(* Logix 5000 project; controller WWTP_SEC_CLX vendor 1 type 14 code 54 rev 17.2; software revision 17.00; part 8 of 13 *)
(* tags used below, declared in another part *)
   Wrk_FirstColdStartT : TIMER;   // Time since first cold start
   Wrk_FirstFailColdT : TIMER;   // Time for cold motor to wait after 1st start failure before ready
   Wrk_SubsFailColdT : TIMER;   // Time for cold motor to wait after 2nd and subs. failures before ready
   Wrk_FirstFailHotT : TIMER;   // Time for hot motor to wait after 1st start failure before ready
   Wrk_SubsFailHotT : TIMER;   // Time for hot motor to wait after 2nd and subs. failures before ready
   Wrk_HotRestartOKT : TIMER;   // Time for hot motor to run so it can restart immediately when stopped
   Wrk_RestartHotT : TIMER;   // Time for hot motor to wait after stop after running less than Hot Restart OK time
   Wrk_HotToColdT : TIMER;   // Time for a stopped hot motor to become cold
   Wrk_State : DINT;   // Instruction State (see state diagram in design docs)
   Wrk_SecondColdStartT : TIMER;   // Time since second cold start
(* P_ResInh, continued *)

ROUTINE Prescan   (* ladder *)
// Clear timers and set to known state
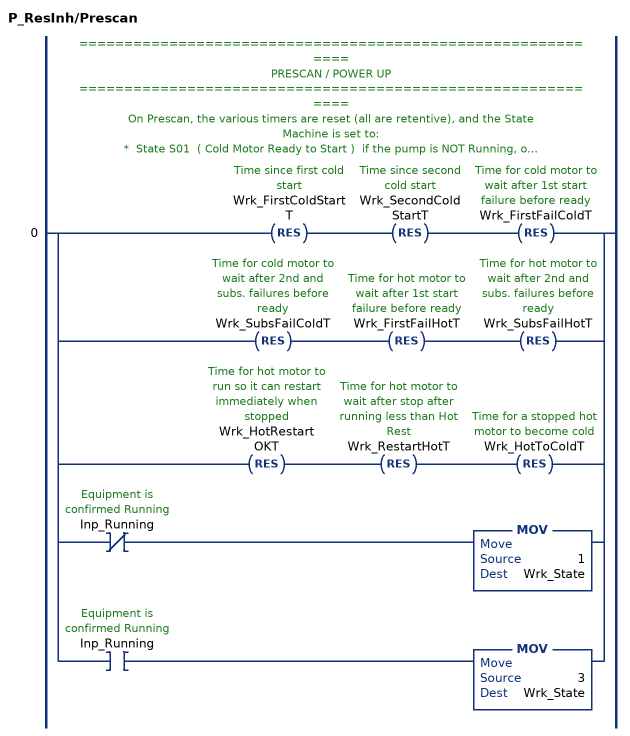
   // ============================================================
   // PRESCAN / POWER UP
   // ============================================================
   // On Prescan, the various timers are reset (all are retentive), and the State
   // Machine is set to:
   // *  State S01  ( Cold Motor Ready to Start )  if the pump is NOT Running, or
   // *  State S03  ( Cold Motor Running )  if the pump is Running.
   0: [RES(Wrk_FirstColdStartT) RES(Wrk_SecondColdStartT) RES(Wrk_FirstFailColdT) ,RES(Wrk_SubsFailColdT) RES(Wrk_FirstFailHotT) RES(Wrk_SubsFailHotT) ,RES(Wrk_HotRestartOKT) RES(Wrk_RestartHotT) RES(Wrk_HotToColdT) ,XIO(Inp_Running) MOV(1,Wrk_State) ,XIC(Inp_Running) MOV(3,Wrk_State) ];
END_ROUTINE
END_ADD_ON_INSTRUCTION

ADD_ON_INSTRUCTION P_RunTime   (* revision 0.7, ExecutePrescan, ExecuteEnableInFalse *)
// Run Time and Starts
// Revision note:
// Aligned name, description and local STRING values, sizes, across instructions.
// Help:
// This Instruction monitors the "Running" and "Starting" Status of a motor or other device and  provides:
// *  Total accumulated run time, in 1/10 hour increments (hour meter)
// *  Total number of starts or start attemptes (count)
// *  Maximum continuous run time for any start (hours)
// *  Program and Maintenance Commands to allow clearing of the totals/maximum
VAR_INPUT
   Inp_Starting : BOOL; {visible}   // 1=Motor is Starting (from motor instruction)
   Inp_Running : BOOL := 1; {visible}   // 1=Motor is Running (from motor instruction)
   Cfg_PCmdClear : BOOL := 1;   // 1=Clear Program Commands on receipt 0=Leave Set
   PCmd_ClearStarts : BOOL;   // Program Command to Clear Count of Starts (attempts)
   PCmd_ClearMaxHrs : BOOL;   // Program Command to Clear Maximum (continuous) Run Time for any start
   PCmd_ClearTotHrs : BOOL;   // Program Command to Clear Total Running Time
   MCmd_ClearStarts : BOOL;   // Maintenance Command to Clear Count of Starts (attempts)
   MCmd_ClearMaxHrs : BOOL;   // Maintenance Command to Clear Maximum (continuous) Run Time for any start
   MCmd_ClearTotHrs : BOOL;   // Maintenance Command to Clear Total Running Time
END_VAR
VAR_OUTPUT
   Val_Starts : DINT; {visible}   // Total number of motor starts or attempts
   Val_CurRunHrs : REAL; {visible}   // Current running time this start (hours)
   Val_MaxRunHrs : REAL; {visible}   // Maximum continuous running time for a given start (hours)
   Val_TotRunHrs : REAL; {visible}   // Total accumulated running time (hours)
END_VAR
VAR
   Wrk_CurHours : DINT;   // Whole hours of current run time
   Wrk_CurRunT : TIMER := (PRE := 2147483647);   // Timer for timing current run time
   Wrk_TotTenths : DINT;   // Tenths of hours of total run time
   Wrk_Starts : COUNTER := (PRE := 2147483647);   // Counter for counting motor starts
   Wrk_TotRunT : TIMER := (PRE := 2147483647);   // Retentive timer for timing 0.1 hour total run time
   Wrk_MaxHours : REAL;   // Internal Maximum Run Hours
END_VAR

ROUTINE EnableInFalse   (* ladder *)
// False Rung or Enable In False: as if motor is Stopped
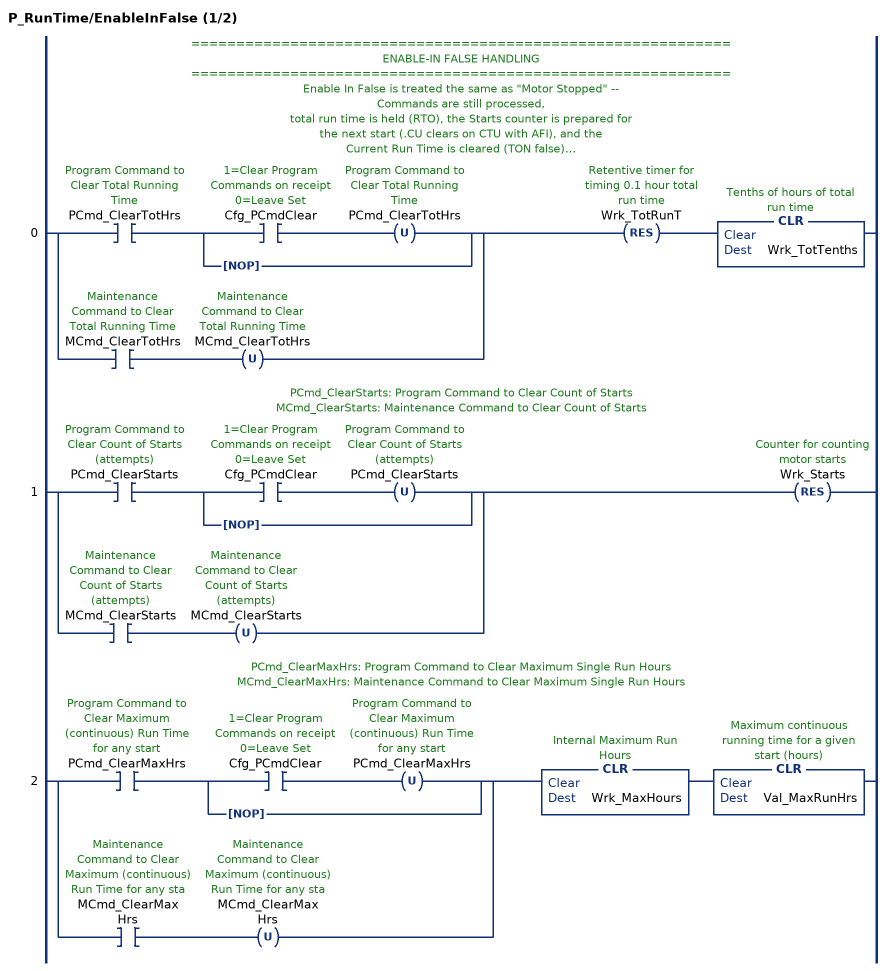
   // ============================================================
   // ENABLE-IN FALSE HANDLING
   // ============================================================
   // Enable In False is treated the same as "Motor Stopped" --
   // Commands are still processed,
   // total run time is held (RTO), the Starts counter is prepared for
   // the next start (.CU clears on CTU with AFI), and the
   // Current Run Time is cleared (TON false).
   // ============================================================
   // COMMAND PROCESSING
   // ============================================================
   // These rungs handle received Commands.  This object has no Modes and
   // Commands are accepted regardless of Mode.  Commands should be
   // restricted to authorized personnel (typically at a maintenance level).
   // PCmd_ClearTotHrs: Program Command to Clear Total Runtime Hours
   // MCmd_ClearTotHrs: Maintenance Command to Clear Total Runtime Hours
   0: [XIC(PCmd_ClearTotHrs) [XIC(Cfg_PCmdClear) OTU(PCmd_ClearTotHrs) ,NOP() ] ,XIC(MCmd_ClearTotHrs) OTU(MCmd_ClearTotHrs) ]RES(Wrk_TotRunT)CLR(Wrk_TotTenths);
   // PCmd_ClearStarts: Program Command to Clear Count of Starts
   // MCmd_ClearStarts: Maintenance Command to Clear Count of Starts
   1: [XIC(PCmd_ClearStarts) [XIC(Cfg_PCmdClear) OTU(PCmd_ClearStarts) ,NOP() ] ,XIC(MCmd_ClearStarts) OTU(MCmd_ClearStarts) ]RES(Wrk_Starts);
   // PCmd_ClearMaxHrs: Program Command to Clear Maximum Single Run Hours
   // MCmd_ClearMaxHrs: Maintenance Command to Clear Maximum Single Run Hours
   2: [XIC(PCmd_ClearMaxHrs) [XIC(Cfg_PCmdClear) OTU(PCmd_ClearMaxHrs) ,NOP() ] ,XIC(MCmd_ClearMaxHrs) OTU(MCmd_ClearMaxHrs) ]CLR(Wrk_MaxHours)CLR(Val_MaxRunHrs);
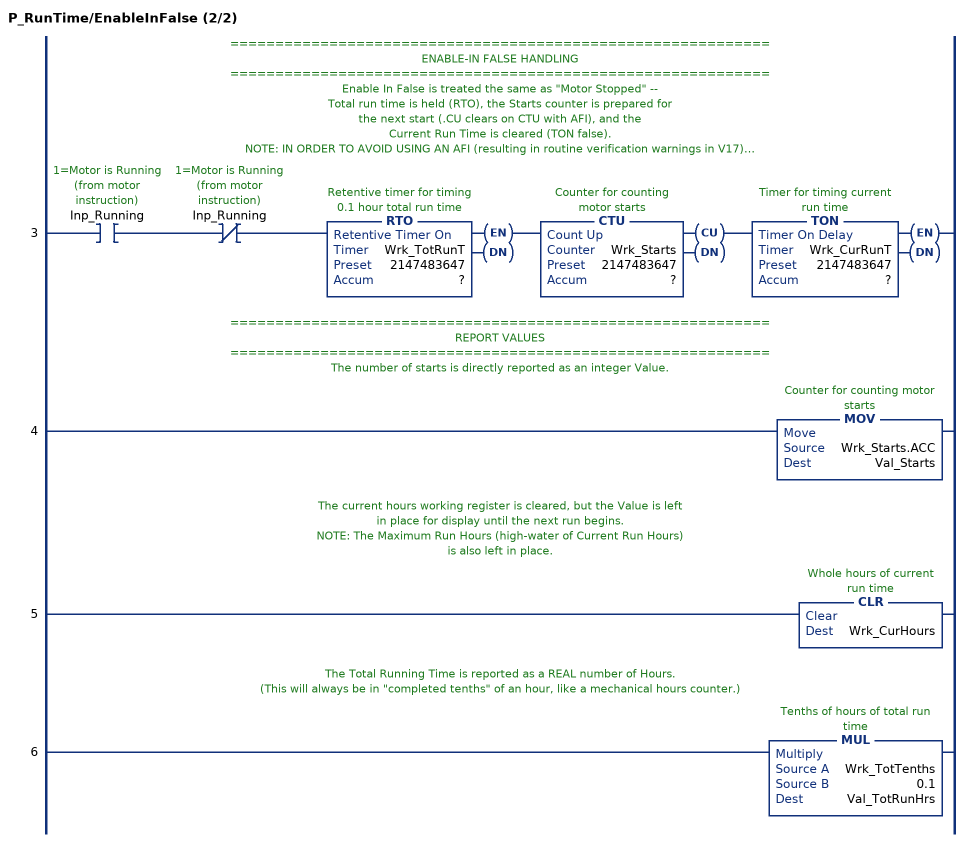
   // ============================================================
   // ENABLE-IN FALSE HANDLING
   // ============================================================
   // Enable In False is treated the same as "Motor Stopped" --
   // Total run time is held (RTO), the Starts counter is prepared for
   // the next start (.CU clears on CTU with AFI), and the
   // Current Run Time is cleared (TON false).
   // NOTE: IN ORDER TO AVOID USING AN AFI (resulting in routine verification warnings in V17),
   // THIS RUNG USES AN XIC AND XIO OF THE SAME BIT TO ENSURE THE
   // TIMERS AND COUNTER ARE SCANNED FALSE.
   // THIS IS NOT DEAD CODE.  IT IS INTENTIONALLY CODED THIS WAY FOR PROPER OPERATION.
   3: XIC(Inp_Running)XIO(Inp_Running)RTO(Wrk_TotRunT,?,?)CTU(Wrk_Starts,?,?)TON(Wrk_CurRunT,?,?);
   // ============================================================
   // REPORT VALUES
   // ============================================================
   // The number of starts is directly reported as an integer Value.
   4: MOV(Wrk_Starts.ACC,Val_Starts);
   // The current hours working register is cleared, but the Value is left
   // in place for display until the next run begins.
   // NOTE: The Maximum Run Hours (high-water of Current Run Hours)
   // is also left in place.
   5: CLR(Wrk_CurHours);
   // The Total Running Time is reported as a REAL number of Hours.
   // (This will always be in "completed tenths" of an hour, like a mechanical hours counter.)
   6: MUL(Wrk_TotTenths,0.1,Val_TotRunHrs);
END_ROUTINE

ROUTINE Logic   (* ladder *)
// Accumulate Run Time (if runnings) and Count Starts
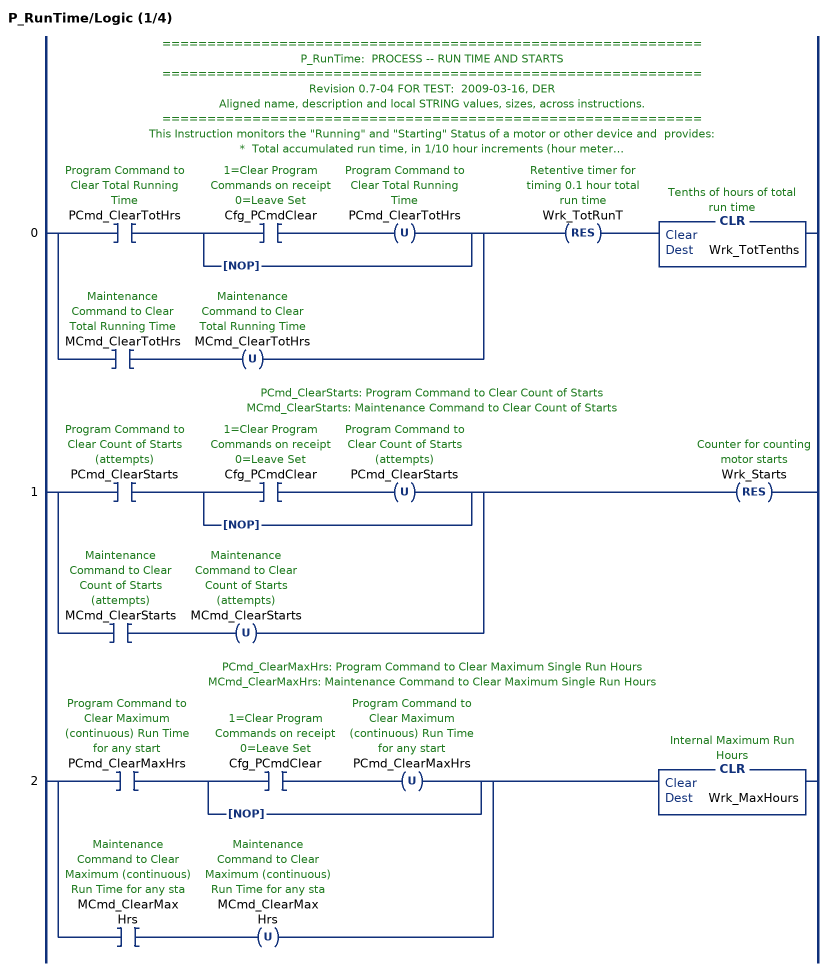
   // ============================================================
   // P_RunTime:  PROCESS -- RUN TIME AND STARTS
   // ============================================================
   // Revision 0.7-04 FOR TEST:  2009-03-16, DER
   // Aligned name, description and local STRING values, sizes, across instructions.
   // ============================================================
   // This Instruction monitors the "Running" and "Starting" Status of a motor or other device and  provides:
   // *  Total accumulated run time, in 1/10 hour increments (hour meter)
   // *  Total number of starts or start attemptes (count)
   // *  Maximum continuous run time for any start (hours)
   // * Commands to allow clearing of the totals/maximum
   // ============================================================
   // COMMAND PROCESSING
   // ============================================================
   // These rungs handle received Commands.  This object has no Modes and
   // Commands are accepted regardless of Mode.  Commands should be
   // restriceted to authorized personnel (typically at a maintenance level).
   // PCmd_ClearTotHrs: Program Command to Clear Total Runtime Hours
   // MCmd_ClearTotHrs: Maintenance Command to Clear Total Runtime Hours
   0: [XIC(PCmd_ClearTotHrs) [XIC(Cfg_PCmdClear) OTU(PCmd_ClearTotHrs) ,NOP() ] ,XIC(MCmd_ClearTotHrs) OTU(MCmd_ClearTotHrs) ]RES(Wrk_TotRunT)CLR(Wrk_TotTenths);
   // PCmd_ClearStarts: Program Command to Clear Count of Starts
   // MCmd_ClearStarts: Maintenance Command to Clear Count of Starts
   1: [XIC(PCmd_ClearStarts) [XIC(Cfg_PCmdClear) OTU(PCmd_ClearStarts) ,NOP() ] ,XIC(MCmd_ClearStarts) OTU(MCmd_ClearStarts) ]RES(Wrk_Starts);
   // PCmd_ClearMaxHrs: Program Command to Clear Maximum Single Run Hours
   // MCmd_ClearMaxHrs: Maintenance Command to Clear Maximum Single Run Hours
   2: [XIC(PCmd_ClearMaxHrs) [XIC(Cfg_PCmdClear) OTU(PCmd_ClearMaxHrs) ,NOP() ] ,XIC(MCmd_ClearMaxHrs) OTU(MCmd_ClearMaxHrs) ]CLR(Wrk_MaxHours);
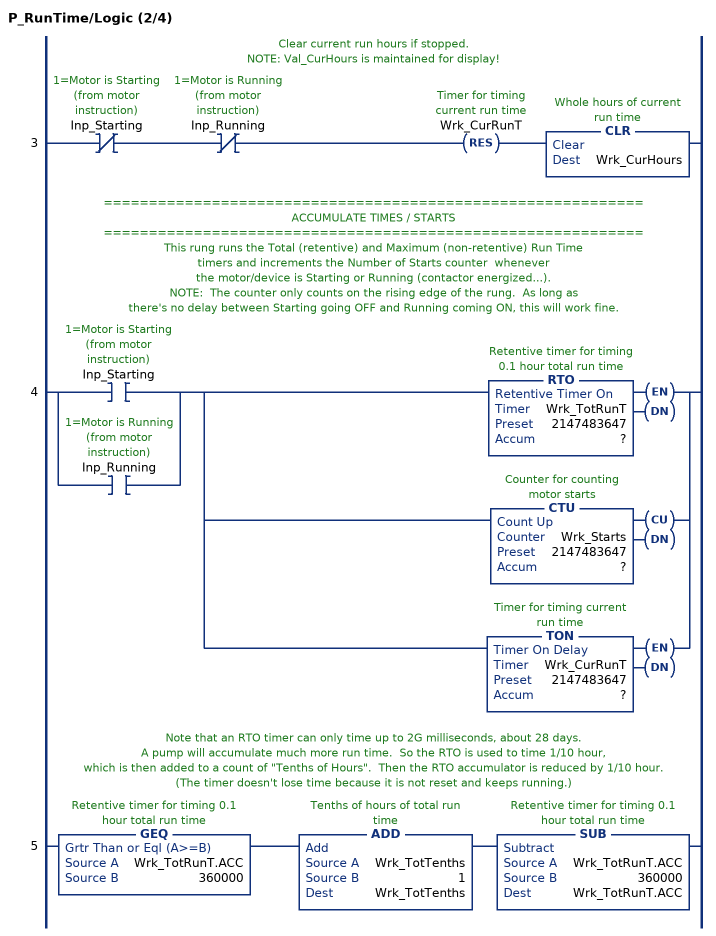
   // Clear current run hours if stopped.
   // NOTE: Val_CurHours is maintained for display!
   3: XIO(Inp_Starting)XIO(Inp_Running)RES(Wrk_CurRunT)CLR(Wrk_CurHours);
   // ============================================================
   // ACCUMULATE TIMES / STARTS
   // ============================================================
   // This rung runs the Total (retentive) and Maximum (non-retentive) Run Time
   // timers and increments the Number of Starts counter  whenever
   //  the motor/device is Starting or Running (contactor energized...).
   // NOTE:  The counter only counts on the rising edge of the rung.  As long as
   // there's no delay between Starting going OFF and Running coming ON, this will work fine.
   4: [XIC(Inp_Starting) ,XIC(Inp_Running) ][RTO(Wrk_TotRunT,?,?) ,CTU(Wrk_Starts,?,?) ,TON(Wrk_CurRunT,?,?) ];
   // Note that an RTO timer can only time up to 2G milliseconds, about 28 days.
   // A pump will accumulate much more run time.  So the RTO is used to time 1/10 hour,
   // which is then added to a count of "Tenths of Hours".  Then the RTO accumulator is reduced by 1/10 hour.
   // (The timer doesn't lose time because it is not reset and keeps running.)
   5: GEQ(Wrk_TotRunT.ACC,360000)ADD(Wrk_TotTenths,1,Wrk_TotTenths)SUB(Wrk_TotRunT.ACC,360000,Wrk_TotRunT.ACC);
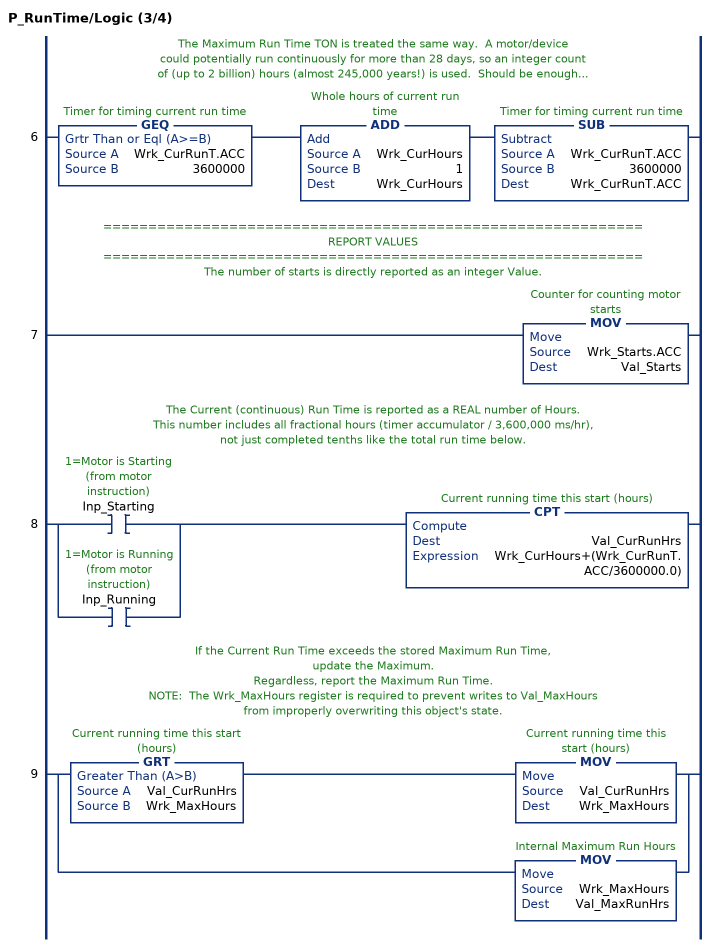
   // The Maximum Run Time TON is treated the same way.  A motor/device
   // could potentially run continuously for more than 28 days, so an integer count
   // of (up to 2 billion) hours (almost 245,000 years!) is used.  Should be enough...
   6: GEQ(Wrk_CurRunT.ACC,3600000)ADD(Wrk_CurHours,1,Wrk_CurHours)SUB(Wrk_CurRunT.ACC,3600000,Wrk_CurRunT.ACC);
   // ============================================================
   // REPORT VALUES
   // ============================================================
   // The number of starts is directly reported as an integer Value.
   7: MOV(Wrk_Starts.ACC,Val_Starts);
   // The Current (continuous) Run Time is reported as a REAL number of Hours.
   // This number includes all fractional hours (timer accumulator / 3,600,000 ms/hr),
   // not just completed tenths like the total run time below.
   8: [XIC(Inp_Starting) ,XIC(Inp_Running) ]CPT(Val_CurRunHrs,Wrk_CurHours+(Wrk_CurRunT.ACC/3600000.0));
   // If the Current Run Time exceeds the stored Maximum Run Time,
   // update the Maximum.
   // Regardless, report the Maximum Run Time.
   // NOTE:  The Wrk_MaxHours register is required to prevent writes to Val_MaxHours
   // from improperly overwriting this object's state.
   9: [GRT(Val_CurRunHrs,Wrk_MaxHours) MOV(Val_CurRunHrs,Wrk_MaxHours) ,MOV(Wrk_MaxHours,Val_MaxRunHrs) ];
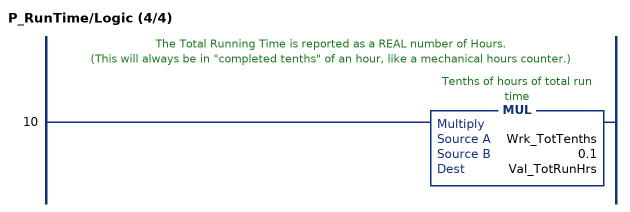
   // The Total Running Time is reported as a REAL number of Hours.
   // (This will always be in "completed tenths" of an hour, like a mechanical hours counter.)
   10: MUL(Wrk_TotTenths,0.1,Val_TotRunHrs);
END_ROUTINE

ROUTINE Prescan   (* ladder *)
// Set Current Run time internally to 0.  Display value is left in place.
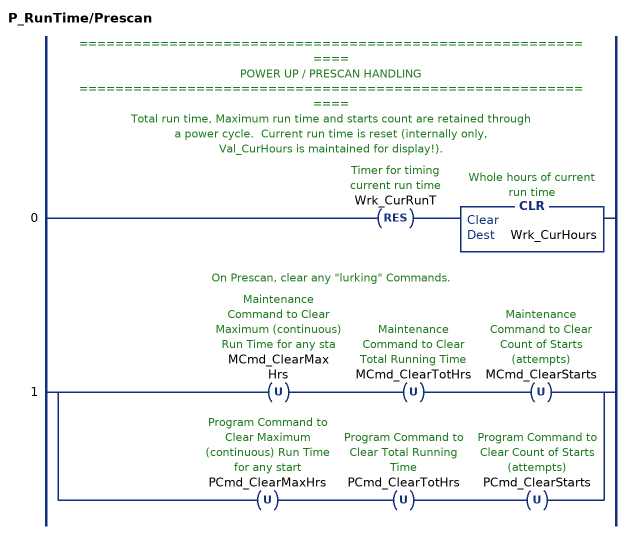
   // ============================================================
   // POWER UP / PRESCAN HANDLING
   // ============================================================
   // Total run time, Maximum run time and starts count are retained through
   // a power cycle.  Current run time is reset (internally only,
   // Val_CurHours is maintained for display!).
   0: RES(Wrk_CurRunT)CLR(Wrk_CurHours);
   // On Prescan, clear any "lurking" Commands.
   1: [OTU(MCmd_ClearMaxHrs) OTU(MCmd_ClearTotHrs) OTU(MCmd_ClearStarts) ,OTU(PCmd_ClearMaxHrs) OTU(PCmd_ClearTotHrs) OTU(PCmd_ClearStarts) ];
END_ROUTINE
END_ADD_ON_INSTRUCTION

ADD_ON_INSTRUCTION P_VSD   (* revision 0.15, ExecutePrescan, ExecuteEnableInFalse *)
// Variable Speed Drive
// Revision note:
// Aligned name, description and local STRING values, sizes, across instructions.
// Help:
// This Instruction controls and monitors a Variable-Speed (AC or DC) Drive
// and provides:
// *  Starting drive, stopping drive, jogging drive, setting speed reference and setting direction
// *  Monitoring of run feedback, display of actual drive status, including accel, decel, direction, speed
// *  Detection of Failure to Start, Failure to Stop, Drive Fault/Not Ready
// *  Monitoring of Permissive conditions to allow starting
// *  Monitoring of Interlock conditions to stop drive or prevent starting
// *  Simulation, providing feedback of a working drive while disabling outputs
// *  Monitoring of I/O communication faults
// *  Alarms for Fail to Start, Fail to Stop, Interlock Trip, Drive Fault/Not Ready, I/O Fault
// *  Operation in Hand, Maintenance, Override, Program and Operator Modes
// *  "Available" status for use by automation logic to know whether drive
//       can be controlled by other objects.
VAR_INPUT
   Inp_SpeedFdbk : INT; {visible}   // Speed Feedbak in Drive Units (typ. 0-32767 = 0 to max freq.)
   Inp_FaultCode : INT;   // Current Drive Fault Code (enumeration)
   Inp_Datalink : INT; {visible}   // Auxiliary Signal (datalink) Input in Drive (raw) Units
   Inp_Ready : BOOL := 1; {visible}   // 1=Drive is ready to run
   Inp_Running : BOOL; {visible}   // 1=Drive is Running (active)
   Inp_CommandDir : BOOL := 1; {visible}   // 1=Drive is commanded Forward, 0=Drive is commanded Reverse
   Inp_ActualDir : BOOL := 1; {visible}   // 1=Drive is running Forward, 0=Drive is running Reverse
   Inp_Accelerating : BOOL; {visible}   // 1=Drive is accelerating
   Inp_Decelerating : BOOL; {visible}   // 1=Drive is decelerating
   Inp_Alarm : BOOL; {visible}   // 1=Drive has an Alarm Condition (see drive display or manual)
   Inp_Faulted : BOOL; {visible}   // 1=Drive has Faulted (see drive display or manual)
   Inp_AtSpeed : BOOL; {visible}   // 1=Drive is at commanded speed
   Inp_FwdPermOK : BOOL := 1; {visible}   // 1=Permissives OK, drive can start Forward
   Inp_FwdNBPermOK : BOOL := 1; {visible}   // 1=Non-Bypassable Permissives OK, drive can start Forward
   Inp_RevPermOK : BOOL := 1; {visible}   // 1=Permissives OK, drive can start Reverse
   Inp_RevNBPermOK : BOOL := 1; {visible}   // 1=Non-Bypassable Permissives OK, motor can start Reverse
   Inp_IntlkOK : BOOL := 1; {visible}   // 1=Interlocks OK, drive can start/run
   Inp_NBIntlkOK : BOOL := 1; {visible}   // 1=Non-Bypassable Interlocks OK, drive can start/run
   Inp_IOFault : BOOL;   // Input Communication Status 0=OK, 1=fail
   Inp_Sim : BOOL;   // 1=Simulate working drive; 0=Start/Stop/ Monitor actual drive
   Inp_Hand : BOOL; {visible}   // 1=Select Hand (hardwired) Control Strategy
   Inp_Ovrd : BOOL; {visible}   // 1=Select Override control strategy
   Inp_OvrdState : BOOL; {visible}   // 1=Override to RUN, 0=Override to STOP
   Inp_OvrdSpeed : REAL; {visible}   // Speed at which to run drive in Override if Overriding to RUN
   Inp_Reset : BOOL; {visible}   // 1=Reset drive fault conditions and latched Alarms
   Cfg_HasReverse : BOOL;   // 1=Drive can be run reverse, 0=Forward only
   Cfg_HasJog : BOOL;   // 1=Drive Jog Command enabled/visible, 0=Drive Jog Command not allowed
   Cfg_HasRunFdbk : BOOL := 1;   // 1=Drive provides speed feedback and run signal
   Cfg_UseRunFdbk : BOOL := 1;   // 1=Drive run feedback should be used for failure checking
   Cfg_HasInpDatalink : BOOL;   // 1=A signal is connected to Inp_Datalink1
   Cfg_HasOutDatalink : BOOL;   // 1=A signal is connected to Out_Datalink1
   Cfg_HasFwdPermObj : BOOL;   // 1=Tells HMI a P_Perm is connected to Inp_FwdPerm
   Cfg_HasRevPermObj : BOOL;   // 1=Tells HMI a P_Perm is connected to Inp_RevPerm
   Cfg_HasIntlkObj : BOOL;   // 1=Tells HMI a P_Intlk is connected to Inp_Intlk
   Cfg_HasResInhObj : BOOL;   // 1=Tells HMI a P_ResInh Restart Inhibit is connected
   Cfg_HasRunTimeObj : BOOL;   // 1=Tells HMI a P_RunTime is connected
   Cfg_SetTrack : BOOL := 1;   // 1=PSets track OSets in Oper, OSets track PSets in Prog, 0=no tracking
   Cfg_SetTrackOvrdHand : BOOL;   // 1=Prog/Oper Settings track Override/Hand speed reference
   Cfg_PCmdClear : BOOL := 1;   // 1=Clear Program Commands on receipt 0=Leave Set
   Cfg_OvrdPermIntlk : BOOL;   // 1=Override ignores Bypassable Perm/ Intlk; 0=always use Perm/Intlk
   Cfg_HasFailToStartAlm : BOOL;   // 1=Fail to Start Alarm exists and will be checked
   Cfg_HasFailToStopAlm : BOOL;   // 1=Fail to Stop Alarm exists and will be checked
   Cfg_HasIntlkTripAlm : BOOL;   // 1=Interlock Trip Alarm exists and will be checked
   Cfg_HasDriveFaultAlm : BOOL;   // 1=Drive Fault alarm exists and will be checked
   Cfg_HasIOFaultAlm : BOOL;   // 1=I/O Fault Alarm exists and will be checked
   Cfg_FailToStartResetReqd : BOOL;   // 1=Reset requied to clear Fail to Start Alarm
   Cfg_FailToStopResetReqd : BOOL;   // 1=Reset required to clear Fail to Stop Alarm
   Cfg_IntlkTripResetReqd : BOOL;   // 1=Reset required to clear Interlock Trip Alarm
   Cfg_DriveFaultResetReqd : BOOL := 1;   // 1=Reset required to clear Drive Fault Alarm
   Cfg_IOFaultResetReqd : BOOL;   // 1=Reset required to clear I/O Fault Alarm
   Cfg_FailToStartAckReqd : BOOL := 1;   // 1=Acknowledge required for Fail to Start Alarm
   Cfg_FailToStopAckReqd : BOOL := 1;   // 1=Acknowledge required for Fail to Stop Alarm
   Cfg_IntlkTripAckReqd : BOOL := 1;   // 1=Acknowledge required for Interlock Trip Alarm
   Cfg_DriveFaultAckReqd : BOOL;   // 1=Acknowledge required for Drive Fault Alarm
   Cfg_IOFaultAckReqd : BOOL := 1;   // 1=Acknowledge required for I/O Fault Alarm
   Cfg_FailToStartSeverity : SINT := 4;   // Fail To Start Alarm Severity 1=info 2=warn 3=excep 4=fault
   Cfg_FailToStopSeverity : SINT := 4;   // Fail To Stop Alarm Severity 1=info 2=warn 3=excep 4=fault
   Cfg_IntlkTripSeverity : SINT := 2;   // Interlock Trip Alarm Severity 1=info 2=warn 3=excep 4=fault
   Cfg_DriveFaultSeverity : SINT := 4;   // Drive Fault Alarm Severity 1=info, 2=warn, 3=excep, 4=fault
   Cfg_IOFaultSeverity : SINT := 4;   // I/O Fault Alarm Severity 1=info 2=warn 3=excep 4=fault
   Cfg_MinSpdRef : REAL;   // Minimum Speed Reference in EU (for limiting)
   Cfg_MaxSpdRef : REAL := 60.0;   // Maximum Speed Reference in EU (for limiting)
   Cfg_SpeedRefRawMin : INT;   // Speed Reference Minimum in Drive (raw) Units (for scaling)
   Cfg_SpeedRefRawMax : INT := 32767;   // Speed Reference Maximum in Drive (raw) Units (for scaling)
   Cfg_SpeedRefEUMin : REAL;   // Speed Reference Minimum in Engineering Units (for scaling)
   Cfg_SpeedRefEUMax : REAL := 130.0;   // Speed Reference Maximum in Engineering Units (for scaling)
   Cfg_SpeedFdbkRawMin : INT;   // Speed Feedback Minimum in Drive (raw) Units (for scaling)
   Cfg_SpeedFdbkRawMax : INT := 32767;   // Speed Feedback Maximum in Drive (raw) Units (for scaling)
   Cfg_SpeedFdbkEUMin : REAL;   // Speed Feedback Minimum in Engineering Units (for scaling)
   Cfg_SpeedFdbkEUMax : REAL := 130.0;   // Speed Feedback Maximum in Engineering Units (for scaling)
   Cfg_InpDatalinkRawMin : INT;   // Input Datalink Minimum in Drive (raw) Units (for scaling)
   Cfg_InpDatalinkRawMax : INT := 4095;   // Input Datalink Maximum in Drive (raw) Units (for scaling)
   Cfg_InpDatalinkEUMin : REAL;   // Input Datalink Minimum in Engineering Units (for scaling)
   Cfg_InpDatalinkEUMax : REAL := 409.5;   // Input Datalink Maximum in Engineering Units (for scaling)
   Cfg_OutDatalinkMin : REAL;   // Minimum Output Datalink in EU (for limiting)
   Cfg_OutDatalinkMax : REAL := 100.0;   // Maximum Output Datalink in EU (for limiting)
   Cfg_OutDatalinkRawMin : INT;   // Output Datalink Minimum in Drive (raw) Units (for scaling)
   Cfg_OutDatalinkRawMax : INT := 4095;   // Output Datalink Maximum in Drive (raw) Units (for scaling)
   Cfg_OutDatalinkEUMin : REAL;   // Output Datalink Minimum in Engineering Units (for scaling)
   Cfg_OutDatalinkEUMax : REAL := 409.5;   // Output Datalink Maximum in Engineering Units (for scaling)
   Cfg_SimRampT : DINT := 10;   // Time to ramp speed fdbk when in Simulation (sec)
   Cfg_FailToStartT : DINT := 15;   // Time after Start to get Run Feedback before Fault (sec)
   Cfg_FailToStopT : DINT := 15;   // Time after Stop to drop Run Feedback before Fault (sec)
   Cfg_ResetPulseT : DINT := 2;   // Time to pulse Out_Reset to clear drive fault
   PSet_SpeedRef : REAL;   // Program Setting of Speed Reference (EU)
   PSet_OutDatalink : REAL;   // Program Setting of Output Datalink (EU)
   PSet_Owner : DINT;   // Program Owner Request ID (non-zero) or Release (zero)
   OSet_SpeedRef : REAL;   // Operator Setting of Speed Reference (EU)
   OSet_OutDatalink : REAL;   // Operator Setting of Output Datalink (EU)
   PCmd_Start : BOOL;   // Program Command to Start Drive
   PCmd_Stop : BOOL;   // Program Command to Stop Drive
   PCmd_Fwd : BOOL;   // Program Command to set direction to Fowrard
   PCmd_Rev : BOOL;   // Program Command to set direction to Reverse
   PCmd_Acq : BOOL;   // Program Command to Acquire ownership (Oper/OOS to Prog)
   PCmd_Rel : BOOL;   // Program Command to Release ownership (Prog to OOS)
   PCmd_Lock : BOOL;   // Program Command to Lock Mode in Prog
   PCmd_Unlock : BOOL;   // Program Command to Unlock Mode
   PCmd_Reset : BOOL;   // Program Command to Reset drive fault and all Alarms requiring Reset
   PCmd_FailToStartAck : BOOL;   // Program Command to Acknowledge Fail to Start Alarm
   PCmd_FailToStartInhibit : BOOL;   // Program Command to Inhibit Fail to Start Alarm
   PCmd_FailToStartUninhibit : BOOL;   // Program Command to Uninhibit Fail to Start Alarm
   PCmd_FailToStopAck : BOOL;   // Program Command to Acknowledge Fail to Stop Alarm
   PCmd_FailToStopInhibit : BOOL;   // Program Command to Inhibit Fail to Stop Alarm
   PCmd_FailToStopUninhibit : BOOL;   // Program Command to Uninhibit Fail to Stop Alarm
   PCmd_IntlkTripAck : BOOL;   // Program Command to Acknowledge Interlock Trip Alarm
   PCmd_IntlkTripInhibit : BOOL;   // Program Command to Inhibit Interlock Trip Alarm
   PCmd_IntlkTripUninhibit : BOOL;   // Program Command to Uninhibit Interlock Trip Alarm
   PCmd_DriveFaultAck : BOOL;   // Program Command to Acknowledge Drive Fault Alarm
   PCmd_DriveFaultInhibit : BOOL;   // Program Command to Inhibit Drive Fault Alarm
   PCmd_DriveFaultUninhibit : BOOL;   // Program Command to Uninhibit Drive Fault Alarm
   PCmd_IOFaultAck : BOOL;   // Program Command to Acknowledge I/O Fault Alarm
   PCmd_IOFaultInhibit : BOOL;   // Program Command to Inhibit I/O Fault Alarm
   PCmd_IOFaultUninhibit : BOOL;   // Program Command to Uninhibit I/O Fault Alarm
   OCmd_Start : BOOL;   // Operator Command to Start Drive
   OCmd_Stop : BOOL;   // Operator Command to Stop Drive
   OCmd_Jog : BOOL;   // Operator Command to Jog Drive (not cleared by P_VSD!)
   OCmd_Fwd : BOOL;   // Operator Command to set direction to Forward
   OCmd_Rev : BOOL;   // Operator Command to set direction to Reverse
   OCmd_Bypass : BOOL;   // Operator Command to Bypass all Bypassable Interlocks and Permissives
   OCmd_Check : BOOL;   // Operator Command to Check (not bypass) all Interlocks and Permissives
   MCmd_Disable : BOOL;   // Maintenance Command to Disable Drive
   MCmd_Enable : BOOL;   // Maintenance Command to Enable (allow to run) Drive
   OCmd_Reset : BOOL;   // Operator Command to Reset all Alarms requiring Reset
END_VAR
VAR_OUTPUT
   Out_SpeedRef : INT; {visible}   // Drive Speed Reference in Drive Units (typ. 0-32767 = 0 to max freq.)
   Out_Datalink : INT; {visible}   // Auxiliary Signal (datalink) Output in Drive (raw) Units
   Out_Run : BOOL;   // 1=Start/Run Drive, 0=Stop Drive (for held starter type)
   Out_Stop : BOOL; {visible}   // 1=Stop Drive, 0=drive left in current state
   Out_Start : BOOL; {visible}   // 1=Start Drive, 0=drive left in current state
   Out_Jog : BOOL; {visible}   // 1=Jog drive at Jog Speed, -->0=stop jogging
   Out_ClearFault : BOOL; {visible}   // 1=Attempt to clear Drive Fault
   Out_Fwd : BOOL; {visible}   // 1=Set drive direction to Forward
   Out_Rev : BOOL; {visible}   // 1=Set drive direction to Reverse
   Val_SpeedRef : REAL; {visible}   // Speed Reference (target) to drive
   Val_SpeedFdbk : REAL; {visible}   // Speed Feedback (actual) from drive
   Val_InpDatalink : REAL; {visible}   // Input Datalink value from drive
   Val_OutDatalink : REAL; {visible}   // Output Datalink value to drive
   Val_SpeedFdbkEUMin : REAL;   // Minimum of Speed Feedback = MIN (Cfg_SpeedFdbkEUMin, Cfg_SpeedFdbkEUMax)
   Val_SpeedFdbkEUMax : REAL := 130.0;   // Maximum of Speed Feedback = MAX (Cfg_SpeedFdbkEUMin, Cfg_SpeedFdbkEUMax)
   Val_Owner : DINT;   // Current Object Owner ID (0=not owned)
   Val_Notify : SINT;   // Current Alarm Level and Acknowledgement (enumeration)
   Sts_Stopped : BOOL := 1; {visible}   // 1=Drive requested to stop and is confirmed stopped
   Sts_Starting : BOOL; {visible}   // 1=Drive requested to run and awaiting run feedback
   Sts_Running : BOOL; {visible}   // 1=Drive requested to run and is confirmed running
   Sts_Stopping : BOOL; {visible}   // 1=Drive requested to stop and awaiting stopped feedback
   Sts_Jogging : BOOL; {visible}   // 1=Drive requested to Jog
   Sts_CommandDir : BOOL := 1;   // 1=Drive commanded to Forward, 0=Reverse
   Sts_ActualDir : BOOL := 1; {visible}   // 1=Drive Actual direction is Forward, 0=Reverse
   Sts_Accel : BOOL;   // 1=Drive is Accelerating
   Sts_Decel : BOOL;   // 1=Drive is Decelerating
   Sts_NotReady : BOOL; {visible}   // 1=Drive is Not Ready (cannot be started) Check alarms, stops, faults
   Sts_Alarm : BOOL; {visible}   // 1=Drive has an Alarm (see drive display or manual)
   Sts_AtSpeed : BOOL; {visible}   // 1=Drive is running at reference speed
   Sts_SpeedLimited : BOOL; {visible}   // 1=Speed Reference Setting exceeds configured Max/Min limit
   Sts_Available : BOOL;   // 1=Drive available for control by automation (Prog)
   Sts_Bypass : BOOL;   // 1=Bypassable Interlocks and Permissives are Bypassed
   Sts_Disabled : BOOL;   // 1=Drive is Disabled
   Sts_Err : BOOL; {visible}   // 1=Error in Config: see detail bits for reason
   Err_Timer : BOOL;   // 1=Error in Config: Invalid Check or Reset Pulse Time (use 0 to 2147483)
   Err_Sim : BOOL;   // 1=Error in Config: simulation timer preset: use 0 to 2147483)
   Err_Alarm : BOOL;   // 1=Error in Config: Invalid Alarm Severity
   Err_FdbkRaw : BOOL;   // 1=Erron in Config: Speed Fdbk Raw Min = Max
   Err_FdbkEU : BOOL;   // 1=Error in Config: Speed Fdbk EU Min = Max
   Err_RefLim : BOOL;   // 1=Error in Config: Speed Ref Limit Min > Max
   Err_RefEU : BOOL;   // 1=Error in Config: Speed Ref EU Min = Max
   Err_RefRaw : BOOL;   // 1=Error in Config: Speed Ref Raw Min = Max
   Err_InpDLRaw : BOOL;   // 1=Error in Config: Input Datalink Raw Min = Max
   Err_InpDLEU : BOOL;   // 1=Error in Config: Input Datalink EU Min = Max
   Err_OutDLLim : BOOL;   // 1=Error in Config: Output Datalink Limits Min > Max
   Err_OutDLEU : BOOL;   // 1=Error in Config: Output Datalink EU Min = Max
   Err_OutDLRaw : BOOL;   // 1=Error in Config: Output Datalink Raw Min = Max
   Sts_Hand : BOOL; {visible}   // 1=Mode is Hand (supersedes Maint, Ovrd, Prog, Oper)
   Sts_Maint : BOOL; {visible}   // 1=Mode is Maintenance (supersedes Ovrd, Prog, Oper)
   Sts_Ovrd : BOOL; {visible}   // 1=Mode is Override (supersedes Prog, Oper)
   Sts_Prog : BOOL; {visible}   // 1=Mode is Program (auto)
   Sts_Oper : BOOL := 1; {visible}   // 1=Mode is Operator (manual)
   Sts_ProgOperLock : BOOL;   // 1=Program or Operator has requested Mode Lock
   Sts_FailToStart : BOOL;   // 1=Drive Failed to Start (One-Shot)
   Alm_FailToStart : BOOL;   // 1=Drive Fail to tart Alarm
   Ack_FailToStart : BOOL;   // 1=Fail to Start Alarm has been acknowledged
   Sts_FailToStartDisabled : BOOL;   // 1=Fail to Start Alarm has been disabled (will not be sent)
   Sts_FailToStartInhibited : BOOL;   // 1=Fail to Start Alarm has been inhibited by logic
   Sts_FailToStartSuppressed : BOOL;   // 1=Fail to Start Alarm has been suppressed (logged only)
   Sts_FailToStop : BOOL;   // 1=Drive Failed to Stop
   Alm_FailToStop : BOOL;   // 1=Drive Fail to Stop Alarm
   Ack_FailToStop : BOOL;   // 1=Fail to Stop Alarm has been acknowledged
   Sts_FailToStopDisabled : BOOL;   // 1=Fail to Stop Alarm has been disabled (will not be sent)
   Sts_FailToStopInhibited : BOOL;   // 1=Fail to Stop Alarm has been inhibited by logic
   Sts_FailToStopSuppressed : BOOL;   // 1=Fail to Stop Alarm has been suppressed (logged only)
   Sts_IntlkTrip : BOOL;   // 1=Drive was stopped by an Interlock NOT OK (One-Shot)
   Alm_IntlkTrip : BOOL;   // 1=Alarm: Drive stopped by an Interlock NOT OK
   Ack_IntlkTrip : BOOL;   // 1=Interlock Trip Alarm has been acknowledged
   Sts_IntlkTripDisabled : BOOL;   // 1=Interlock Trip Alarm is Disabled (not saved or sent)
   Sts_IntlkTripInhibited : BOOL;   // 1=Interlock Trip Alarm has been inhibited by logic
   Sts_IntlkTripSuppressed : BOOL;   // 1=Interlock Trip Alarm has been suppressed (logged only)
   Sts_DriveFault : BOOL;   // 1=Drive Fault (see drive display or manual)
   Alm_DriveFault : BOOL;   // 1=Alarm: Drive Fault (see drive display or manual)
   Ack_DriveFault : BOOL;   // 1=Drive Fault Alarm has been acknowledged
   Sts_DriveFaultDisabled : BOOL;   // 1-=Drive Fault Alarm has been disabled (will not be sent)
   Sts_DriveFaultInhibited : BOOL;   // 1=Drive Fault Alarm has been inhibited by logic
   Sts_DriveFaultSuppressed : BOOL;   // 1-Drive Fault Alarm has been suppressed (logged only)
   Sts_IOFault : BOOL;   // I/O Comm Fault Status (0=OK, 1=Bad)
   Alm_IOFault : BOOL;   // 1=I/O Fault Alarm
   Ack_IOFault : BOOL;   // 1=I/O Fault Alarm has been acknowledged
   Sts_IOFaultDisabled : BOOL;   // 1=I/O Fault Alarm is Disabled (not saved or sent)
   Sts_IOFaultInhibited : BOOL;   // 1=I/O Fault Alarm has been inhibited by logic
   Sts_IOFaultSuppressed : BOOL;   // 1=I/O Fault Alarm has been suppressed (logged only)
   Rdy_Start : BOOL;   // 1=Ready to receive OCmd_Start (enables HMI button)
   Rdy_Stop : BOOL;   // 1=Ready to receive OCmd_Stop (enables HMI button)
   Rdy_Jog : BOOL;   // 1=Ready to receive OCmd_Jog (enables HMI button)
   Rdy_Fwd : BOOL;   // 1=Ready to receive OCmd_Fwd (enabled HMI button)
   Rdy_Rev : BOOL;   // 1=Ready to receive OCmd_Rev (enables HMI button)
   Rdy_Bypass : BOOL;   // 1=Ready to receive OCmd_Bypass (enables HMI button)
   Rdy_Check : BOOL;   // 1=Ready to receive OCmd_Check (enables HMI button)
   Rdy_Disable : BOOL;   // 1=Ready to receive MCmd_Disable (enables HMI button)
   Rdy_Enable : BOOL;   // 1=Ready to receive MCmd_Enable (enables HMI button)
   Rdy_Reset : BOOL;   // 1=Ready to receive OCmd_Reset (enables HMI button)
END_VAR
VAR
   Mode : P_Mode := (Cfg_PCmdClear := 1, Cfg_OvrdOverLock := 1, Sts_Oper := 1, Rdy_Rel := 1, Rdy_AcqLock := 1);   // Drive Mode Selection
   IOFault : P_Alarm := (Inp := 1, Cfg_AckReqd := 1, Cfg_Severity := 3, Ack := 1, Rdy_Disable := 1);   // I/O Fault Alarm
   IntlkTrip : P_Alarm := (Inp := 1, Cfg_AckReqd := 1, Cfg_Severity := 3, Ack := 1, Rdy_Disable := 1);   // Interlock Trip Alarm
   FailToStop : P_Alarm := (Inp := 1, Cfg_AckReqd := 1, Cfg_Severity := 3, Ack := 1, Rdy_Disable := 1);   // Drive Failed to Stop Alarm
   FailToStart : P_Alarm := (Inp := 1, Cfg_AckReqd := 1, Cfg_Severity := 3, Ack := 1, Rdy_Disable := 1);   // Drive Failed to Start Alarm
   Cfg_Tag : STRING_20 := 'P_VSD';   // Tagname for display on HMI
   Cfg_Label : STRING_20 := 'Motor Speed Control';   // Label for graphic symbol displayed on HMI
   Cfg_Desc : STRING_40 := 'Variable Speed Drive';   // Description for display on HMI
   Wrk_Run : BOOL;   // 1=Drive should be "running", 0=should be "stopped"
   Wrk_AccelT : TIMER;   // Simulation Accel Ramp timer until Running at speed
   Wrk_Fault : BOOL;   // 1=any Fault has been detected
   Wrk_DecelT : TIMER;   // Simulation Decel Ramp time until fully stopped
   Wrk_RunFdbk : BOOL;   // Run Feedback based on mode, simulation, etc. 1=running
   Wrk_IntlkTrip : BOOL;   // 1=Interlock Not OK Tripped Running Drive
   Wrk_Notify : DINT;   // Buffer for building Val_Notify
   Wrk_Bypass : BOOL;   // Internal Bypassable Permissives and Interlocks are Bypassed flag
   Wrk_Disabled : BOOL;   // Internal Drive is Disabled
   DriveFault : P_Alarm := (Inp := 1, Cfg_AckReqd := 1, Cfg_Severity := 3, Ack := 1, Rdy_Disable := 1);   // Drive Faulted Alarm
   Cfg_SpeedRefEU : STRING_8 := 'Hz';   // Speed Reference Engineering Units for display on HMI
   Wrk_SpeedRef : REAL;   // Working copy of Speed Reference (for limiting)
   Wrk_Rev : BOOL;   // Working (internal) Direction 1=Reverse 0=Forward (default)
   Wrk_Jog : BOOL;   // 1=Jog Drive, 0=Drive not jogging
   Wrk_ResetT : TIMER;   // Reset Output Pulse Timer
   Wrk_ResetCond : BOOL;   // Any incoming Reset condition is TRUE
   Wrk_ResetONS : BOOL;   // One-Shot to fire Reset Timer to ensure min. output ON time.
   Cfg_SpeedFdbkEU : STRING_8 := 'Hz';   // Speed Feedback Engineering Units for display on HMI
   Cfg_OutDatalinkLabel : STRING_20;   // Datalink Output Label displayed on faceplate
   Cfg_InpDatalinkLabel : STRING_20;   // Datalink Input Label displayed on faceplate
   Cfg_OutDatalinkEU : STRING_8;   // Datalink Output Engineering Units for display on HMI
   Cfg_InpDatalinkEU : STRING_8;   // Datalink Input Engineering Units for display on HMI
   Wrk_OutDatalink : REAL;   // Selected Output Datalink setting
   Cfg_RevText : STRING_16 := 'Reverse';   // Name for Reverse Direction, e.g., "Down", "Reverse"
   Cfg_FwdText : STRING_16 := 'Forward';   // Name for Forward Direction, e.g., "Up", "Forward"
   Wrk_StopT : TIMER;   // Stop Check Timer (for Fail to Stop)
   Wrk_StartT : TIMER;   // Start Check Timer (for Fail to Start)
END_VAR

ROUTINE EnableInFalse   (* ladder *)
// Disabled is asserted; Outputs OFF; Run Status shown but Alarms disabled
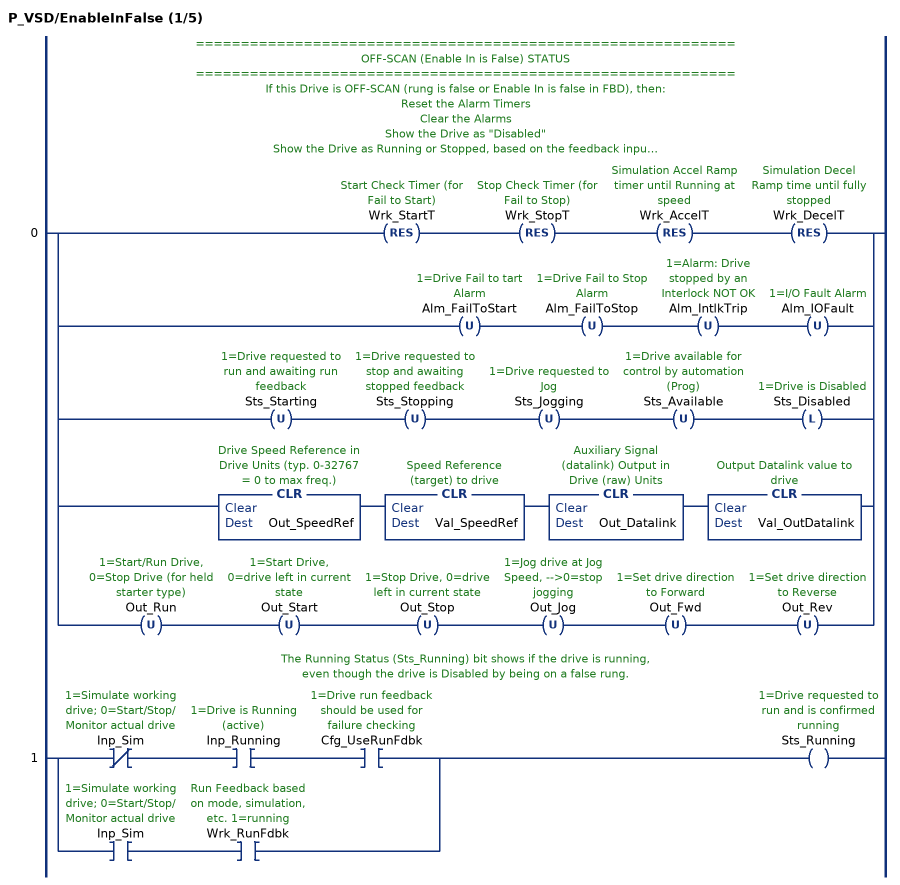
   // ============================================================
   // OFF-SCAN (Enable In is False) STATUS
   // ============================================================
   // If this Drive is OFF-SCAN (rung is false or Enable In is false in FBD), then:
   // Reset the Alarm Timers
   // Clear the Alarms
   // Show the Drive as "Disabled"
   // Show the Drive as Running or Stopped, based on the feedback input
   // Turn off the Outputs, zero the Speed Reference.
   // Other data are left in Last State!
   0: [RES(Wrk_StartT) RES(Wrk_StopT) RES(Wrk_AccelT) RES(Wrk_DecelT) ,OTU(Alm_FailToStart) OTU(Alm_FailToStop) OTU(Alm_IntlkTrip) OTU(Alm_IOFault) ,OTU(Sts_Starting) OTU(Sts_Stopping) OTU(Sts_Jogging) OTU(Sts_Available) OTL(Sts_Disabled) ,CLR(Out_SpeedRef) CLR(Val_SpeedRef) CLR(Out_Datalink) CLR(Val_OutDatalink) ,OTU(Out_Run) OTU(Out_Start) OTU(Out_Stop) OTU(Out_Jog) OTU(Out_Fwd) OTU(Out_Rev) ];
   // The Running Status (Sts_Running) bit shows if the drive is running,
   // even though the drive is Disabled by being on a false rung.
   1: [XIO(Inp_Sim) XIC(Inp_Running) XIC(Cfg_UseRunFdbk) ,XIC(Inp_Sim) XIC(Wrk_RunFdbk) ]OTE(Sts_Running);
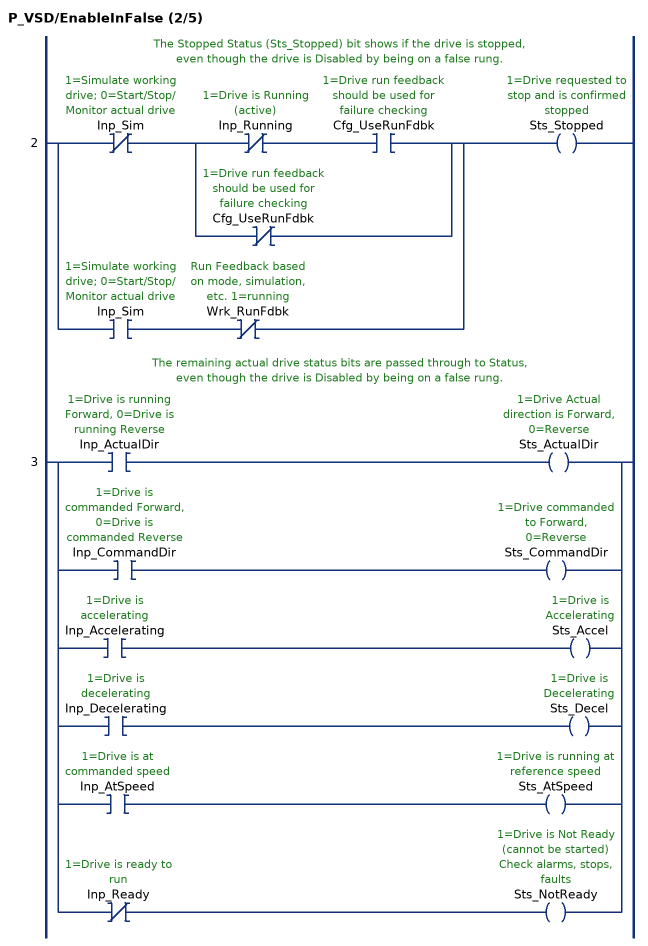
   // The Stopped Status (Sts_Stopped) bit shows if the drive is stopped,
   // even though the drive is Disabled by being on a false rung.
   2: [XIO(Inp_Sim) [XIO(Inp_Running) XIC(Cfg_UseRunFdbk) ,XIO(Cfg_UseRunFdbk) ] ,XIC(Inp_Sim) XIO(Wrk_RunFdbk) ]OTE(Sts_Stopped);
   // The remaining actual drive status bits are passed through to Status,
   // even though the drive is Disabled by being on a false rung.
   3: [XIC(Inp_ActualDir) OTE(Sts_ActualDir) ,XIC(Inp_CommandDir) OTE(Sts_CommandDir) ,XIC(Inp_Accelerating) OTE(Sts_Accel) ,XIC(Inp_Decelerating) OTE(Sts_Decel) ,XIC(Inp_AtSpeed) OTE(Sts_AtSpeed) ,XIO(Inp_Ready) OTE(Sts_NotReady) ];
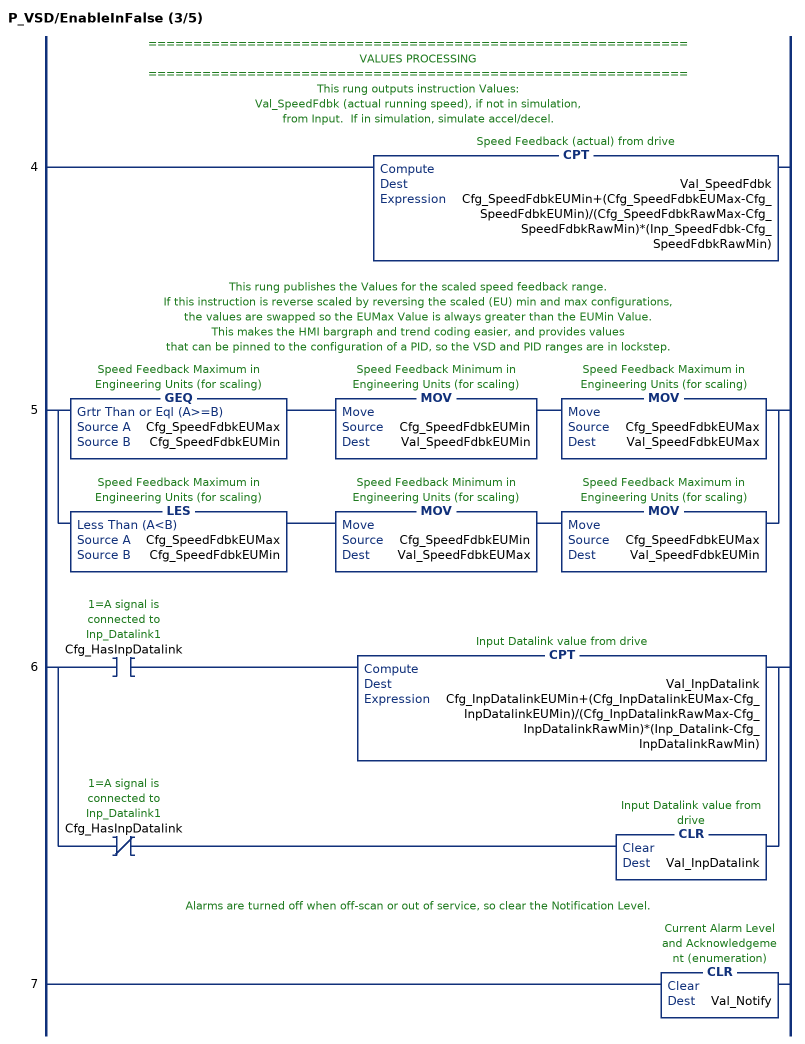
   // ============================================================
   // VALUES PROCESSING
   // ============================================================
   // This rung outputs instruction Values:
   // Val_SpeedFdbk (actual running speed), if not in simulation,
   // from Input.  If in simulation, simulate accel/decel.
   4: CPT(Val_SpeedFdbk,Cfg_SpeedFdbkEUMin+(Cfg_SpeedFdbkEUMax-Cfg_SpeedFdbkEUMin)/(Cfg_SpeedFdbkRawMax-Cfg_SpeedFdbkRawMin)*(Inp_SpeedFdbk-Cfg_SpeedFdbkRawMin));
   // This rung publishes the Values for the scaled speed feedback range.
   // If this instruction is reverse scaled by reversing the scaled (EU) min and max configurations,
   // the values are swapped so the EUMax Value is always greater than the EUMin Value.
   // This makes the HMI bargraph and trend coding easier, and provides values
   // that can be pinned to the configuration of a PID, so the VSD and PID ranges are in lockstep.
   5: [GEQ(Cfg_SpeedFdbkEUMax,Cfg_SpeedFdbkEUMin) MOV(Cfg_SpeedFdbkEUMin,Val_SpeedFdbkEUMin) MOV(Cfg_SpeedFdbkEUMax,Val_SpeedFdbkEUMax) ,LES(Cfg_SpeedFdbkEUMax,Cfg_SpeedFdbkEUMin) MOV(Cfg_SpeedFdbkEUMin,Val_SpeedFdbkEUMax) MOV(Cfg_SpeedFdbkEUMax,Val_SpeedFdbkEUMin) ];
   6: [XIC(Cfg_HasInpDatalink) CPT(Val_InpDatalink,Cfg_InpDatalinkEUMin+(Cfg_InpDatalinkEUMax-Cfg_InpDatalinkEUMin)/(Cfg_InpDatalinkRawMax-Cfg_InpDatalinkRawMin)*(Inp_Datalink-Cfg_InpDatalinkRawMin)) ,XIO(Cfg_HasInpDatalink) CLR(Val_InpDatalink) ];
   // Alarms are turned off when off-scan or out of service, so clear the Notification Level.
   7: CLR(Val_Notify);
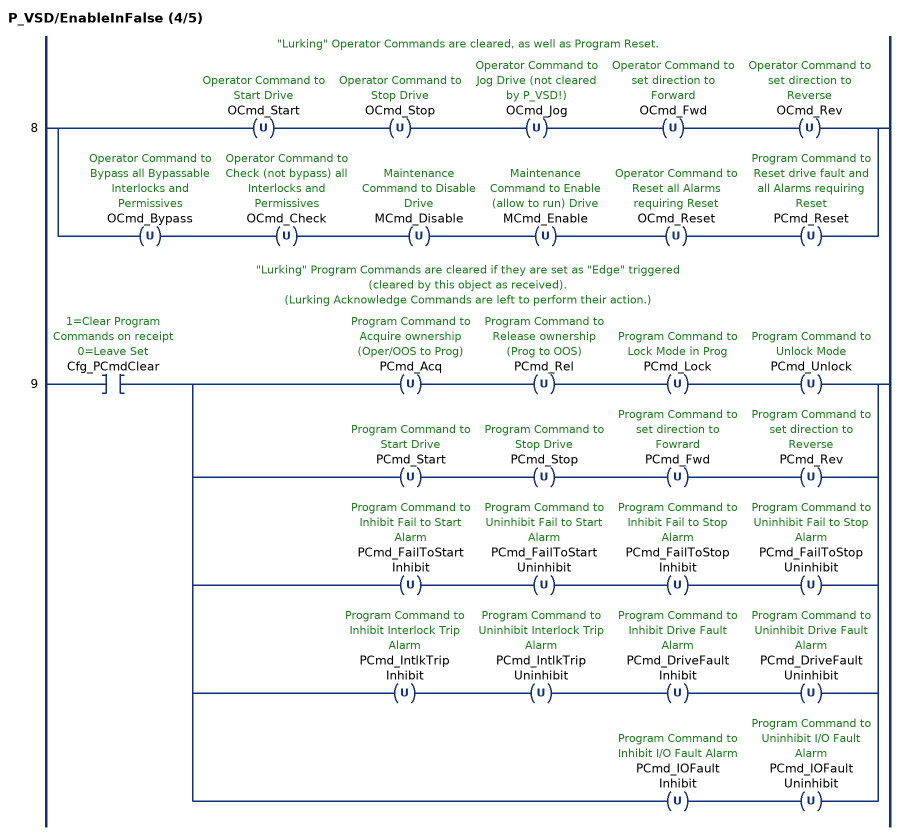
   // "Lurking" Operator Commands are cleared, as well as Program Reset.
   8: [OTU(OCmd_Start) OTU(OCmd_Stop) OTU(OCmd_Jog) OTU(OCmd_Fwd) OTU(OCmd_Rev) ,OTU(OCmd_Bypass) OTU(OCmd_Check) OTU(MCmd_Disable) OTU(MCmd_Enable) OTU(OCmd_Reset) OTU(PCmd_Reset) ];
   // "Lurking" Program Commands are cleared if they are set as "Edge" triggered
   // (cleared by this object as received).
   // (Lurking Acknowledge Commands are left to perform their action.)
   9: XIC(Cfg_PCmdClear)[OTU(PCmd_Acq) OTU(PCmd_Rel) OTU(PCmd_Lock) OTU(PCmd_Unlock) ,OTU(PCmd_Start) OTU(PCmd_Stop) OTU(PCmd_Fwd) OTU(PCmd_Rev) ,OTU(PCmd_FailToStartInhibit) OTU(PCmd_FailToStartUninhibit) OTU(PCmd_FailToStopInhibit) OTU(PCmd_FailToStopUninhibit) ,OTU(PCmd_IntlkTripInhibit) OTU(PCmd_IntlkTripUninhibit) OTU(PCmd_DriveFaultInhibit) OTU(PCmd_DriveFaultUninhibit) ,OTU(PCmd_IOFaultInhibit) OTU(PCmd_IOFaultUninhibit) ];
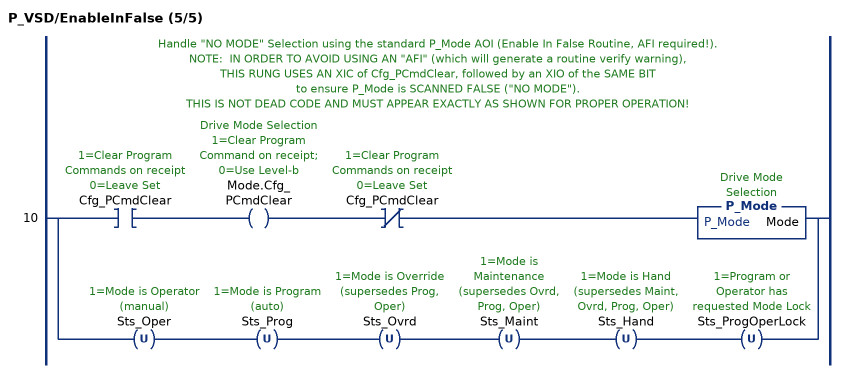
   // Handle "NO MODE" Selection using the standard P_Mode AOI (Enable In False Routine, AFI required!).
   // NOTE:  IN ORDER TO AVOID USING AN "AFI" (which will generate a routine verify warning),
   // THIS RUNG USES AN XIC of Cfg_PCmdClear, followed by an XIO of the SAME BIT
   // to ensure P_Mode is SCANNED FALSE ("NO MODE").
   // THIS IS NOT DEAD CODE AND MUST APPEAR EXACTLY AS SHOWN FOR PROPER OPERATION!
   10: [XIC(Cfg_PCmdClear) OTE(Mode.Cfg_PCmdClear) XIO(Cfg_PCmdClear) P_Mode(Mode) ,OTU(Sts_Oper) OTU(Sts_Prog) OTU(Sts_Ovrd) OTU(Sts_Maint) OTU(Sts_Hand) OTU(Sts_ProgOperLock) ];
END_ROUTINE

ROUTINE Logic   (* ladder *)
// Normal Scan: control / monitor Variable-Speed Drive
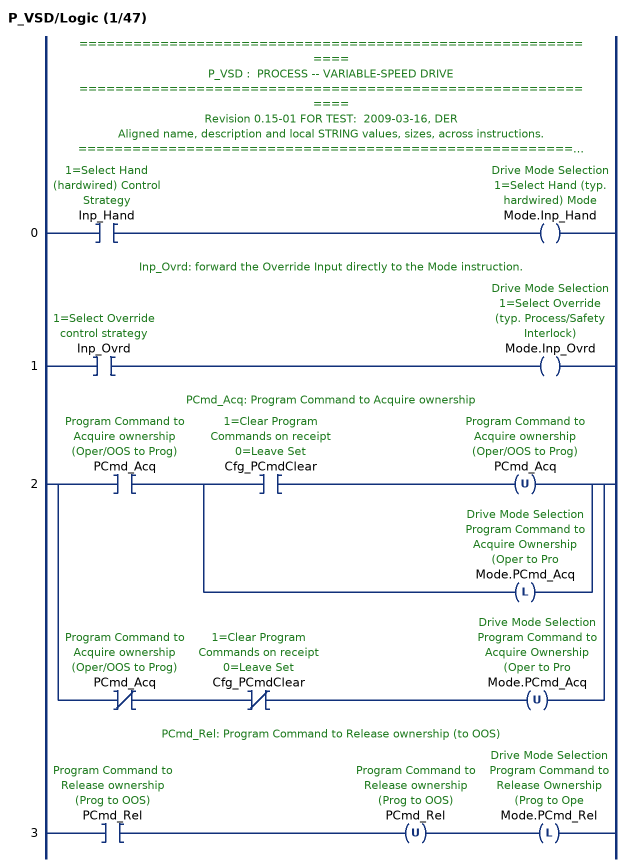
   // ============================================================
   // P_VSD :  PROCESS -- VARIABLE-SPEED DRIVE
   // ============================================================
   // Revision 0.15-01 FOR TEST:  2009-03-16, DER
   // Aligned name, description and local STRING values, sizes, across instructions.
   // ============================================================
   // This Instruction controls and monitors a Variable-Speed Drive (AC or DC) and provides:
   // *  Starting, stopping, jogging of drive, setting speed reference and direction
   // *  Monitoring of run feedback, display of actual drive status, including accel, decel, direction, speed
   // *  Detection of Failure to Start, Failure to Stop, Drive Fault
   // *  Monitoring of Permissive conditions to allow starting
   // * Monitoring of Interlock conditions to stop / prevent starting
   // * Simulation, providing feedback of a working drive while disabling outputs
   // * Monitoring of I/O communication faults
   // * Alarms for Fail to Start, Fail to Stop, Interlock Trip, Drive Fault, I/O Fault
   // * Operation in Hand, Maintenance, Override, Program and Operator Modes
   // * "Available" status for use by automation logic to know whether Drive
   // can be controlled by other objects.
   // ============================================================
   // POWER UP / INVALID STATE HANDLING
   // ============================================================
   // Mode states are retained through a power cycle.
   // Drive "run" request is cleared on first scan, in the rung which unlatches "Wrk_Run", below
   // ============================================================
   // MODE PROCESSING
   // ============================================================
   // These rungs handle received Mode Inputs and Commands:
   // NOTE:  Operator Commands for Mode, Alarm are sent directly to the contained P_Mode and P_Alarm AOIs.
   // Inp_Hand: forward the Hand Input directly to the Mode instruction.
   0: XIC(Inp_Hand)OTE(Mode.Inp_Hand);
   // Inp_Ovrd: forward the Override Input directly to the Mode instruction.
   1: XIC(Inp_Ovrd)OTE(Mode.Inp_Ovrd);
   // PCmd_Acq: Program Command to Acquire ownership
   2: [XIC(PCmd_Acq) [XIC(Cfg_PCmdClear) OTU(PCmd_Acq) ,OTL(Mode.PCmd_Acq) ] ,XIO(PCmd_Acq) XIO(Cfg_PCmdClear) OTU(Mode.PCmd_Acq) ];
   // PCmd_Rel: Program Command to Release ownership (to OOS)
   3: XIC(PCmd_Rel)OTU(PCmd_Rel)OTL(Mode.PCmd_Rel);
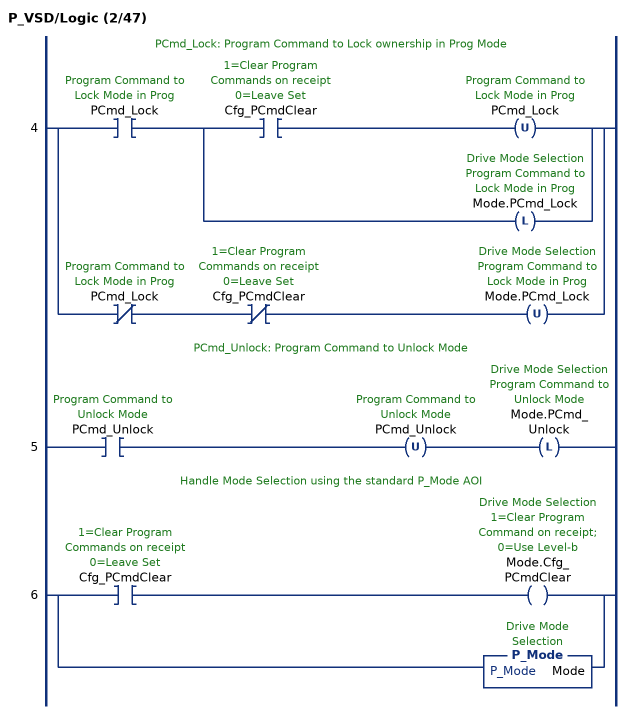
   // PCmd_Lock: Program Command to Lock ownership in Prog Mode
   4: [XIC(PCmd_Lock) [XIC(Cfg_PCmdClear) OTU(PCmd_Lock) ,OTL(Mode.PCmd_Lock) ] ,XIO(PCmd_Lock) XIO(Cfg_PCmdClear) OTU(Mode.PCmd_Lock) ];
   // PCmd_Unlock: Program Command to Unlock Mode
   5: XIC(PCmd_Unlock)OTU(PCmd_Unlock)OTL(Mode.PCmd_Unlock);
   // Handle Mode Selection using the standard P_Mode AOI
   6: [XIC(Cfg_PCmdClear) OTE(Mode.Cfg_PCmdClear) ,P_Mode(Mode) ];
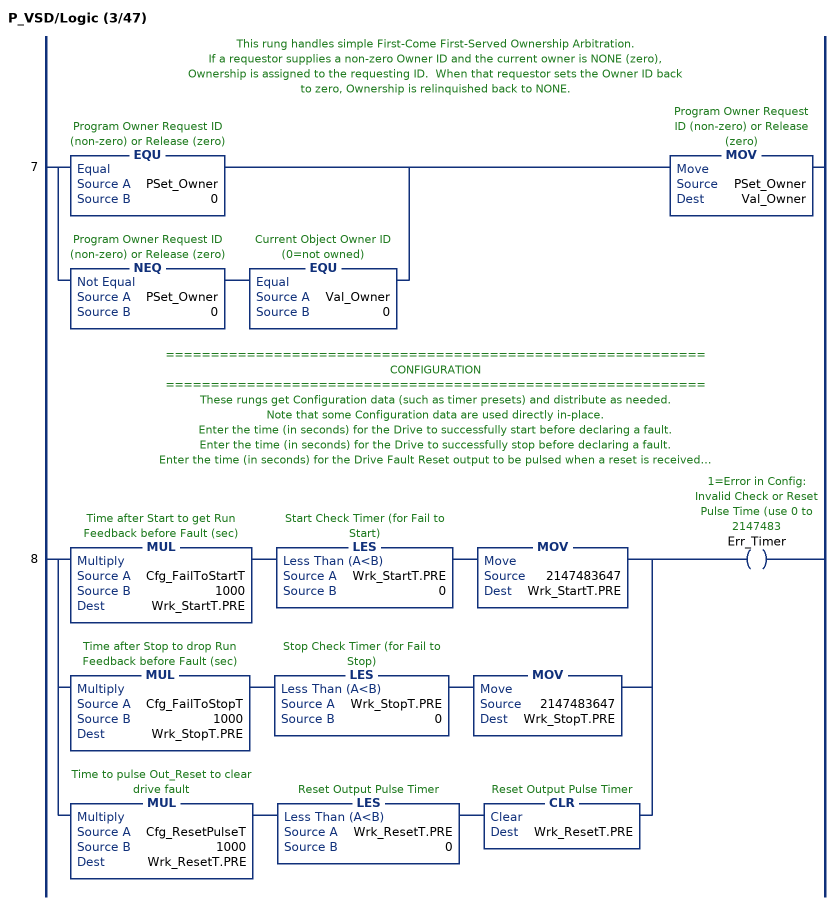
   // This rung handles simple First-Come First-Served Ownership Arbitration.
   // If a requestor supplies a non-zero Owner ID and the current owner is NONE (zero),
   // Ownership is assigned to the requesting ID.  When that requestor sets the Owner ID back
   // to zero, Ownership is relinquished back to NONE.
   7: [EQU(PSet_Owner,0) ,NEQ(PSet_Owner,0) EQU(Val_Owner,0) ]MOV(PSet_Owner,Val_Owner);
   // ============================================================
   // CONFIGURATION
   // ============================================================
   // These rungs get Configuration data (such as timer presets) and distribute as needed.
   // Note that some Configuration data are used directly in-place.
   // Enter the time (in seconds) for the Drive to successfully start before declaring a fault.
   // Enter the time (in seconds) for the Drive to successfully stop before declaring a fault.
   // Enter the time (in seconds) for the Drive Fault Reset output to be pulsed when a reset is received.
   // If the timer preset calculated wraps negative (more than 2.14... million seconds), then max out the
   // or clear the Timer Preset (as appropriate) and flag it.  Note that a negative timer preset will fault the controller!!!
   8: [MUL(Cfg_FailToStartT,1000,Wrk_StartT.PRE) LES(Wrk_StartT.PRE,0) MOV(2147483647,Wrk_StartT.PRE) ,MUL(Cfg_FailToStopT,1000,Wrk_StopT.PRE) LES(Wrk_StopT.PRE,0) MOV(2147483647,Wrk_StopT.PRE) ,MUL(Cfg_ResetPulseT,1000,Wrk_ResetT.PRE) LES(Wrk_ResetT.PRE,0) CLR(Wrk_ResetT.PRE) ]OTE(Err_Timer);
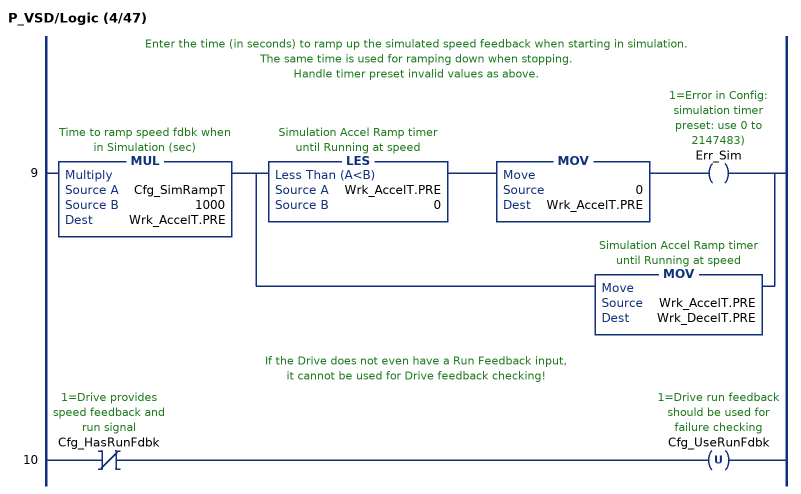
   // Enter the time (in seconds) to ramp up the simulated speed feedback when starting in simulation.
   // The same time is used for ramping down when stopping.
   // Handle timer preset invalid values as above.
   9: MUL(Cfg_SimRampT,1000,Wrk_AccelT.PRE)[LES(Wrk_AccelT.PRE,0) MOV(0,Wrk_AccelT.PRE) OTE(Err_Sim) ,MOV(Wrk_AccelT.PRE,Wrk_DecelT.PRE) ];
   // If the Drive does not even have a Run Feedback input,
   // it cannot be used for Drive feedback checking!
   10: XIO(Cfg_HasRunFdbk)OTU(Cfg_UseRunFdbk);
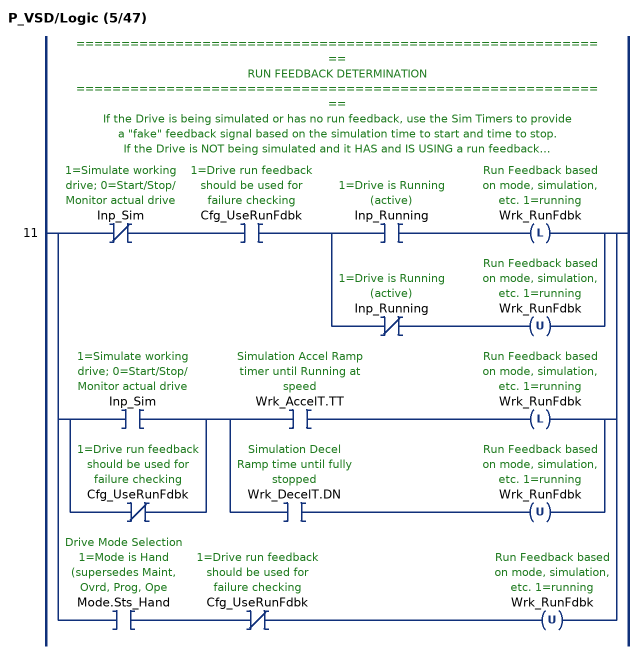
   // ============================================================
   // RUN FEEDBACK DETERMINATION
   // ============================================================
   // If the Drive is being simulated or has no run feedback, use the Sim Timers to provide
   // a "fake" feedback signal based on the simulation time to start and time to stop.
   // If the Drive is NOT being simulated and it HAS and IS USING a run feedback,
   // use the state of the run feedback input as the Drive run state.
   11: [XIO(Inp_Sim) XIC(Cfg_UseRunFdbk) [XIC(Inp_Running) OTL(Wrk_RunFdbk) ,XIO(Inp_Running) OTU(Wrk_RunFdbk) ] ,[XIC(Inp_Sim) ,XIO(Cfg_UseRunFdbk) ] [XIC(Wrk_AccelT.TT) OTL(Wrk_RunFdbk) ,XIC(Wrk_DecelT.DN) OTU(Wrk_RunFdbk) ] ,XIC(Mode.Sts_Hand) XIO(Cfg_UseRunFdbk) OTU(Wrk_RunFdbk) ];
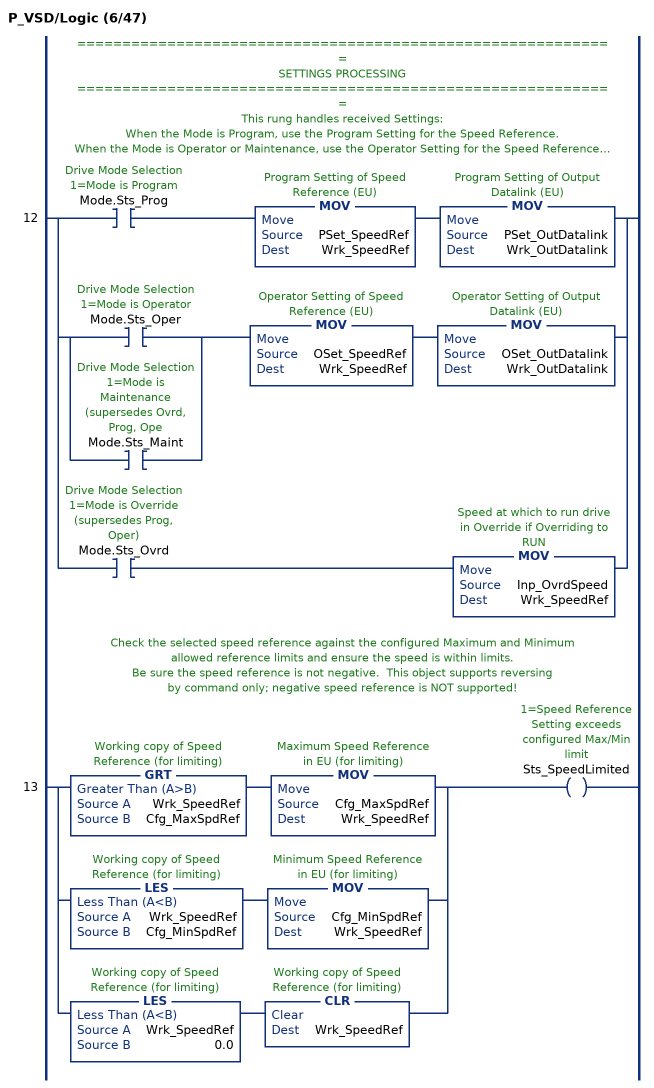
   // ============================================================
   // SETTINGS PROCESSING
   // ============================================================
   // This rung handles received Settings:
   // When the Mode is Program, use the Program Setting for the Speed Reference.
   // When the Mode is Operator or Maintenance, use the Operator Setting for the Speed Reference.
   // When the Mode is Override, use the Override Speed Reference input.
   12: [XIC(Mode.Sts_Prog) MOV(PSet_SpeedRef,Wrk_SpeedRef) MOV(PSet_OutDatalink,Wrk_OutDatalink) ,[XIC(Mode.Sts_Oper) ,XIC(Mode.Sts_Maint) ] MOV(OSet_SpeedRef,Wrk_SpeedRef) MOV(OSet_OutDatalink,Wrk_OutDatalink) ,XIC(Mode.Sts_Ovrd) MOV(Inp_OvrdSpeed,Wrk_SpeedRef) ];
   // Check the selected speed reference against the configured Maximum and Minimum
   // allowed reference limits and ensure the speed is within limits.
   // Be sure the speed reference is not negative.  This object supports reversing
   // by command only; negative speed reference is NOT supported!
   13: [GRT(Wrk_SpeedRef,Cfg_MaxSpdRef) MOV(Cfg_MaxSpdRef,Wrk_SpeedRef) ,LES(Wrk_SpeedRef,Cfg_MinSpdRef) MOV(Cfg_MinSpdRef,Wrk_SpeedRef) ,LES(Wrk_SpeedRef,0.0) CLR(Wrk_SpeedRef) ]OTE(Sts_SpeedLimited);
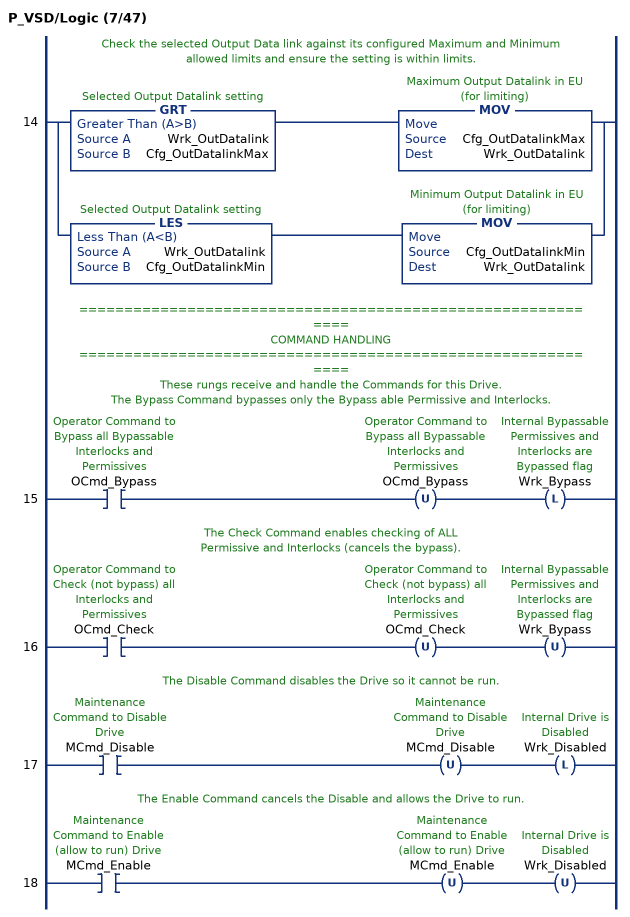
   // Check the selected Output Data link against its configured Maximum and Minimum
   // allowed limits and ensure the setting is within limits.
   14: [GRT(Wrk_OutDatalink,Cfg_OutDatalinkMax) MOV(Cfg_OutDatalinkMax,Wrk_OutDatalink) ,LES(Wrk_OutDatalink,Cfg_OutDatalinkMin) MOV(Cfg_OutDatalinkMin,Wrk_OutDatalink) ];
   // ============================================================
   // COMMAND HANDLING
   // ============================================================
   // These rungs receive and handle the Commands for this Drive.
   // The Bypass Command bypasses only the Bypass able Permissive and Interlocks.
   15: XIC(OCmd_Bypass)OTU(OCmd_Bypass)OTL(Wrk_Bypass);
   // The Check Command enables checking of ALL
   // Permissive and Interlocks (cancels the bypass).
   16: XIC(OCmd_Check)OTU(OCmd_Check)OTU(Wrk_Bypass);
   // The Disable Command disables the Drive so it cannot be run.
   17: XIC(MCmd_Disable)OTU(MCmd_Disable)OTL(Wrk_Disabled);
   // The Enable Command cancels the Disable and allows the Drive to run.
   18: XIC(MCmd_Enable)OTU(MCmd_Enable)OTU(Wrk_Disabled);
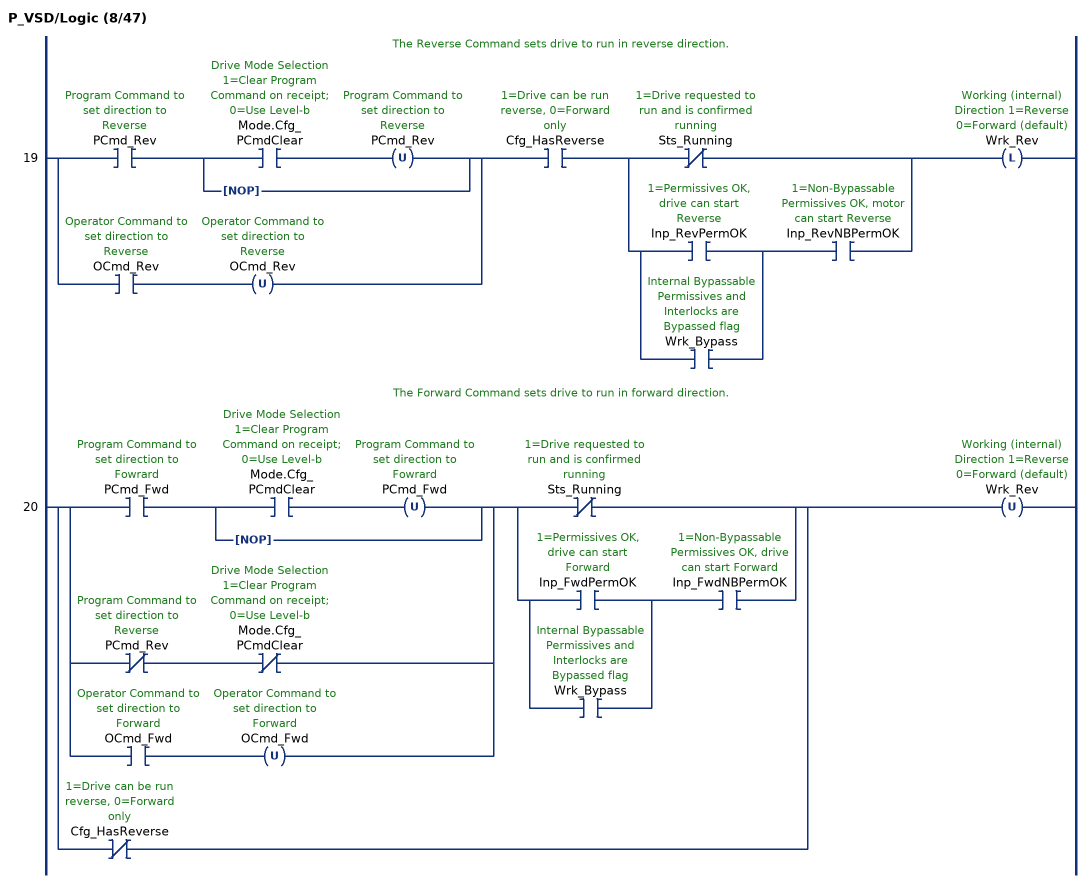
   // The Reverse Command sets drive to run in reverse direction.
   19: [XIC(PCmd_Rev) [XIC(Mode.Cfg_PCmdClear) OTU(PCmd_Rev) ,NOP() ] ,XIC(OCmd_Rev) OTU(OCmd_Rev) ]XIC(Cfg_HasReverse)[XIO(Sts_Running) ,[XIC(Inp_RevPermOK) ,XIC(Wrk_Bypass) ] XIC(Inp_RevNBPermOK) ]OTL(Wrk_Rev);
   // The Forward Command sets drive to run in forward direction.
   20: [[XIC(PCmd_Fwd) [XIC(Mode.Cfg_PCmdClear) OTU(PCmd_Fwd) ,NOP() ] ,XIO(PCmd_Rev) XIO(Mode.Cfg_PCmdClear) ,XIC(OCmd_Fwd) OTU(OCmd_Fwd) ] [XIO(Sts_Running) ,[XIC(Inp_FwdPermOK) ,XIC(Wrk_Bypass) ] XIC(Inp_FwdNBPermOK) ] ,XIO(Cfg_HasReverse) ]OTU(Wrk_Rev);
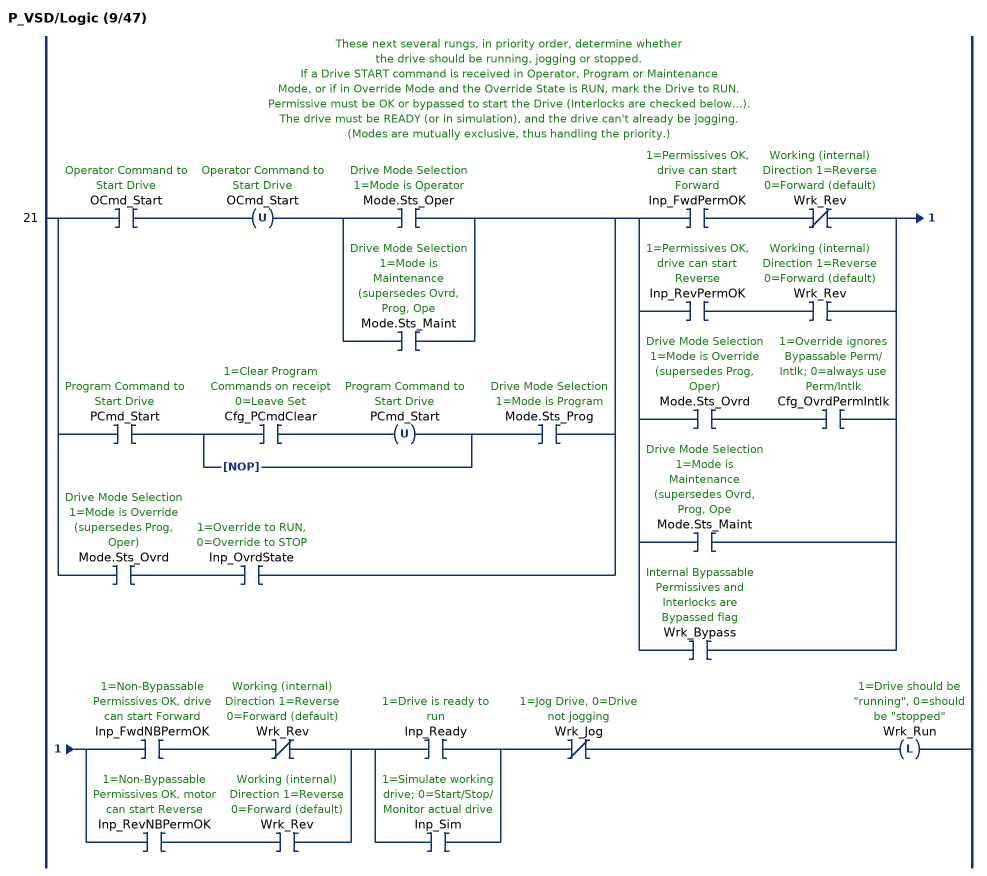
   // These next several rungs, in priority order, determine whether
   // the drive should be running, jogging or stopped.
   // If a Drive START command is received in Operator, Program or Maintenance
   // Mode, or if in Override Mode and the Override State is RUN, mark the Drive to RUN.
   // Permissive must be OK or bypassed to start the Drive (Interlocks are checked below...).
   // The drive must be READY (or in simulation), and the drive can't already be jogging.
   // (Modes are mutually exclusive, thus handling the priority.)
   21: [XIC(OCmd_Start) OTU(OCmd_Start) [XIC(Mode.Sts_Oper) ,XIC(Mode.Sts_Maint) ] ,XIC(PCmd_Start) [XIC(Cfg_PCmdClear) OTU(PCmd_Start) ,NOP() ] XIC(Mode.Sts_Prog) ,XIC(Mode.Sts_Ovrd) XIC(Inp_OvrdState) ][XIC(Inp_FwdPermOK) XIO(Wrk_Rev) ,XIC(Inp_RevPermOK) XIC(Wrk_Rev) ,XIC(Mode.Sts_Ovrd) XIC(Cfg_OvrdPermIntlk) ,XIC(Mode.Sts_Maint) ,XIC(Wrk_Bypass) ][XIC(Inp_FwdNBPermOK) XIO(Wrk_Rev) ,XIC(Inp_RevNBPermOK) XIC(Wrk_Rev) ][XIC(Inp_Ready) ,XIC(Inp_Sim) ]XIO(Wrk_Jog)OTL(Wrk_Run);
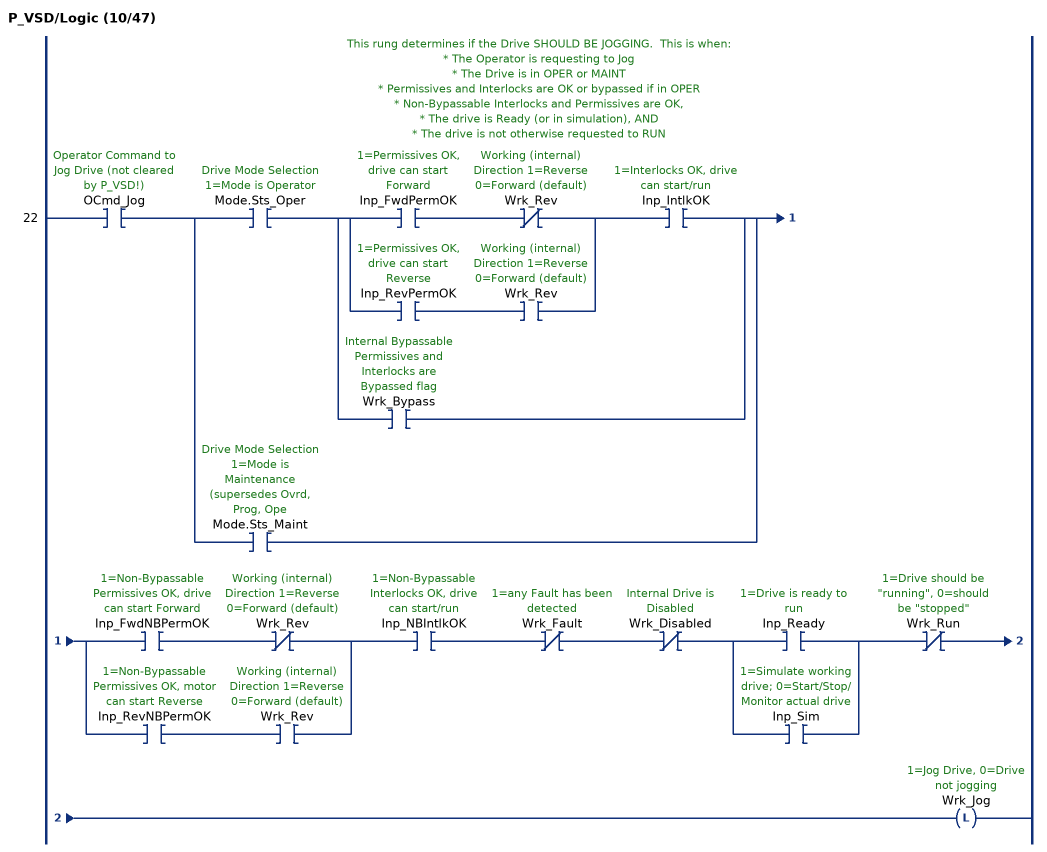
   // This rung determines if the Drive SHOULD BE JOGGING.  This is when:
   // * The Operator is requesting to Jog
   // * The Drive is in OPER or MAINT
   // * Permissives and Interlocks are OK or bypassed if in OPER
   // * Non-Bypassable Interlocks and Permissives are OK,
   // * The drive is Ready (or in simulation), AND
   // * The drive is not otherwise requested to RUN
   22: XIC(OCmd_Jog)[XIC(Mode.Sts_Oper) [[XIC(Inp_FwdPermOK) XIO(Wrk_Rev) ,XIC(Inp_RevPermOK) XIC(Wrk_Rev) ] XIC(Inp_IntlkOK) ,XIC(Wrk_Bypass) ] ,XIC(Mode.Sts_Maint) ][XIC(Inp_FwdNBPermOK) XIO(Wrk_Rev) ,XIC(Inp_RevNBPermOK) XIC(Wrk_Rev) ]XIC(Inp_NBIntlkOK)XIO(Wrk_Fault)XIO(Wrk_Disabled)[XIC(Inp_Ready) ,XIC(Inp_Sim) ]XIO(Wrk_Run)OTL(Wrk_Jog);
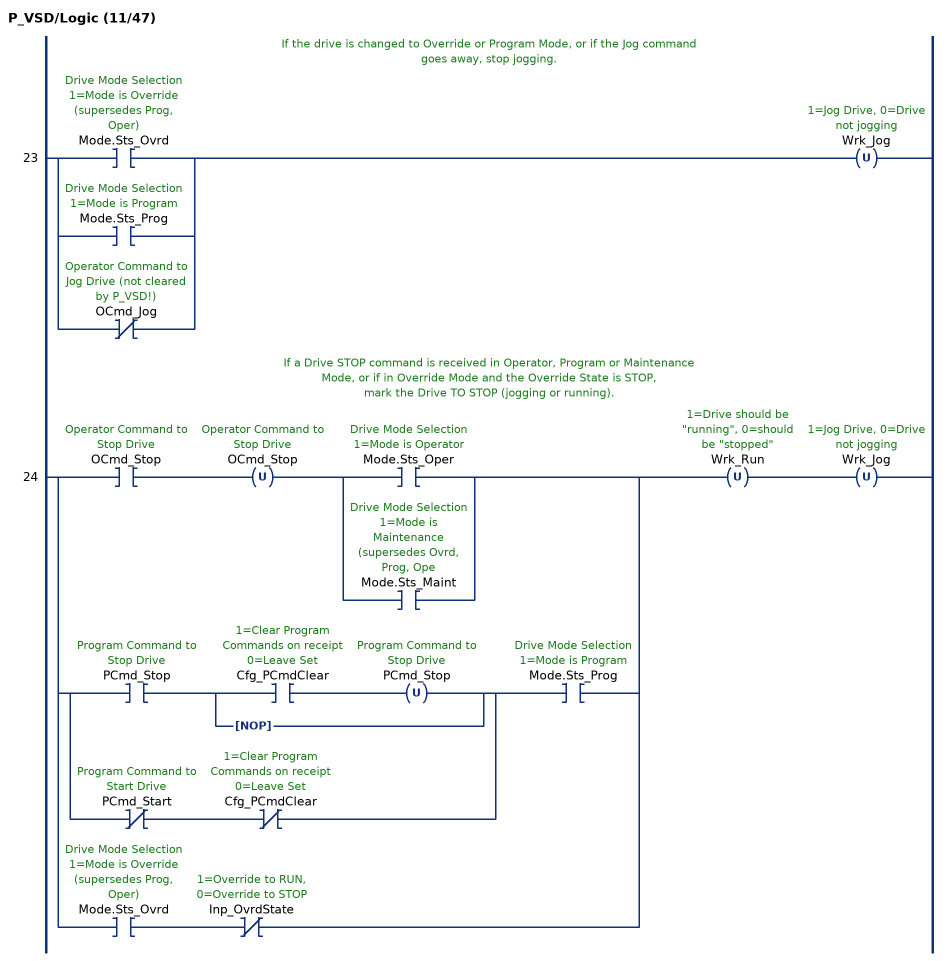
   // If the drive is changed to Override or Program Mode, or if the Jog command
   // goes away, stop jogging.
   23: [XIC(Mode.Sts_Ovrd) ,XIC(Mode.Sts_Prog) ,XIO(OCmd_Jog) ]OTU(Wrk_Jog);
   // If a Drive STOP command is received in Operator, Program or Maintenance
   // Mode, or if in Override Mode and the Override State is STOP,
   // mark the Drive TO STOP (jogging or running).
   24: [XIC(OCmd_Stop) OTU(OCmd_Stop) [XIC(Mode.Sts_Oper) ,XIC(Mode.Sts_Maint) ] ,[XIC(PCmd_Stop) [XIC(Cfg_PCmdClear) OTU(PCmd_Stop) ,NOP() ] ,XIO(PCmd_Start) XIO(Cfg_PCmdClear) ] XIC(Mode.Sts_Prog) ,XIC(Mode.Sts_Ovrd) XIO(Inp_OvrdState) ]OTU(Wrk_Run)OTU(Wrk_Jog);
